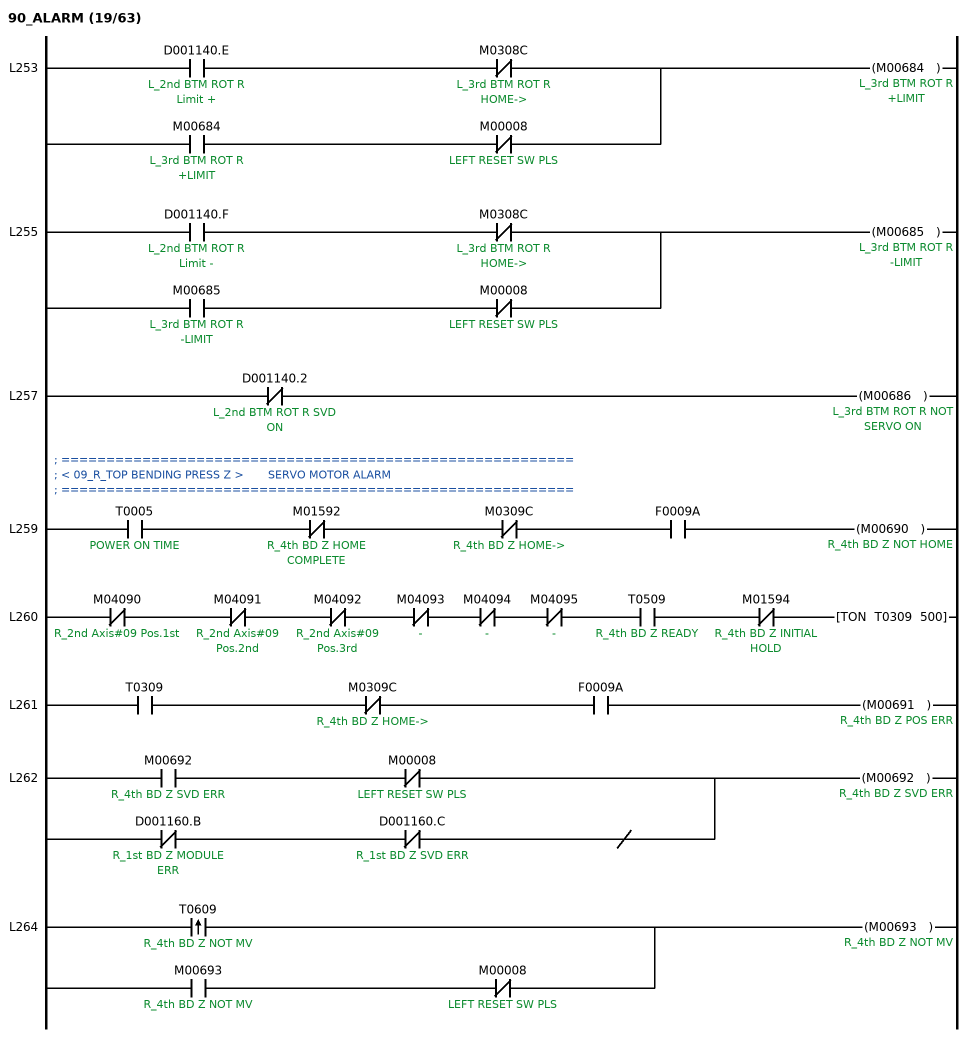
[picture p384: 90_ALARM rungs L253-L264]
; L253
LOAD      D001140.E	// L_2nd BTM ROT R Limit +
AND NOT   M0308C	// L_3rd BTM ROT R HOME->
LOAD      M00684	// L_3rd BTM ROT R +LIMIT
AND NOT   M00008	// LEFT RESET SW PLS
OR LOAD
OUT       M00684	// L_3rd BTM ROT R +LIMIT
; L255
LOAD      D001140.F	// L_2nd BTM ROT R Limit -
AND NOT   M0308C	// L_3rd BTM ROT R HOME->
LOAD      M00685	// L_3rd BTM ROT R -LIMIT
AND NOT   M00008	// LEFT RESET SW PLS
OR LOAD
OUT       M00685	// L_3rd BTM ROT R -LIMIT
; L257
LOAD NOT  D001140.2	// L_2nd BTM ROT R SVD ON
OUT       M00686	// L_3rd BTM ROT R NOT SERVO ON
// =========================================================
// 
//        < 09_R_TOP BENDING PRESS Z >       SERVO MOTOR ALARM
// 
// =========================================================
; L259
LOAD      T0005	// POWER ON TIME
AND NOT   M01592	// R_4th BD Z HOME COMPLETE
AND NOT   M0309C	// R_4th BD Z HOME->
AND       F0009A
OUT       M00690	// R_4th BD Z NOT HOME
; L260
LOAD NOT  M04090	// R_2nd Axis#09 Pos.1st
AND NOT   M04091	// R_2nd Axis#09 Pos.2nd
AND NOT   M04092	// R_2nd Axis#09 Pos.3rd
AND NOT   M04093	// -
AND NOT   M04094	// -
AND NOT   M04095	// -
AND       T0509	// R_4th BD Z READY
AND NOT   M01594	// R_4th BD Z INITIAL HOLD
TON       T0309 500
; L261
LOAD      T0309
AND NOT   M0309C	// R_4th BD Z HOME->
AND       F0009A
OUT       M00691	// R_4th BD Z POS ERR
; L262
LOAD      M00692	// R_4th BD Z SVD ERR
AND NOT   M00008	// LEFT RESET SW PLS
LOAD NOT  D001160.B	// R_1st BD Z MODULE ERR
AND NOT   D001160.C	// R_1st BD Z SVD ERR
NOT
OR LOAD
OUT       M00692	// R_4th BD Z SVD ERR
; L264
LOADP     T0609	// R_4th BD Z NOT MV
LOAD      M00693	// R_4th BD Z NOT MV
AND NOT   M00008	// LEFT RESET SW PLS
OR LOAD
OUT       M00693	// R_4th BD Z NOT MV

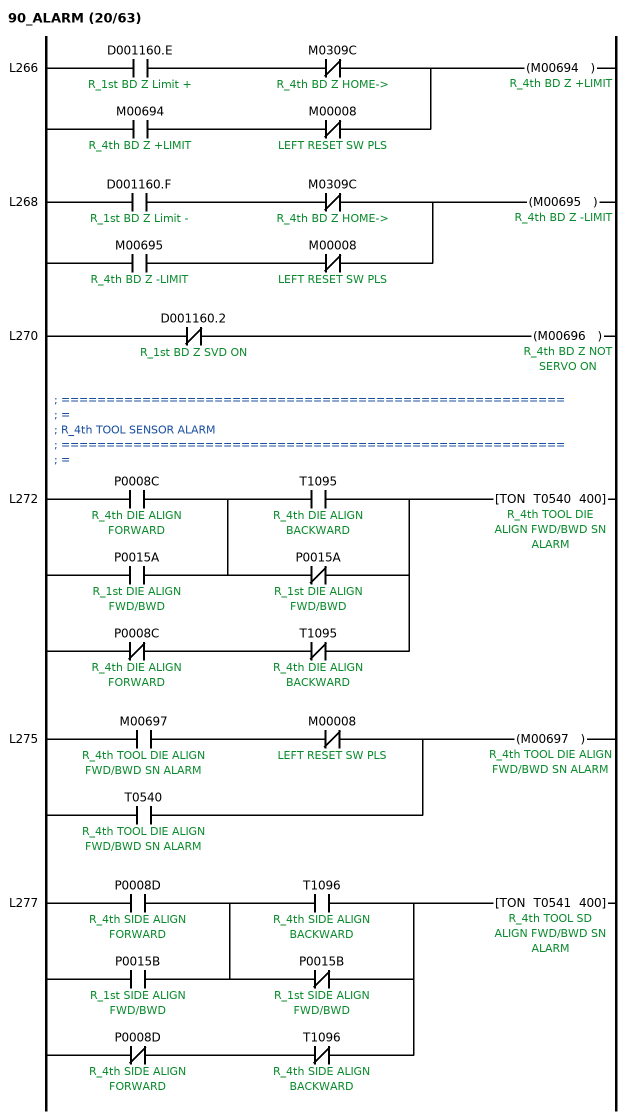
; L266
LOAD      D001160.E	// R_1st BD Z Limit +
AND NOT   M0309C	// R_4th BD Z HOME->
LOAD      M00694	// R_4th BD Z +LIMIT
AND NOT   M00008	// LEFT RESET SW PLS
OR LOAD
OUT       M00694	// R_4th BD Z +LIMIT
; L268
LOAD      D001160.F	// R_1st BD Z Limit -
AND NOT   M0309C	// R_4th BD Z HOME->
LOAD      M00695	// R_4th BD Z -LIMIT
AND NOT   M00008	// LEFT RESET SW PLS
OR LOAD
OUT       M00695	// R_4th BD Z -LIMIT
; L270
LOAD NOT  D001160.2	// R_1st BD Z SVD ON
OUT       M00696	// R_4th BD Z NOT SERVO ON
// =========================================================
// 
//        R_4th TOOL SENSOR ALARM
// 
// =========================================================
; L272
LOAD      P0008C	// R_4th DIE ALIGN FORWARD
OR        P0015A	// R_1st DIE ALIGN FWD/BWD
LOAD      T1095	// R_4th DIE ALIGN BACKWARD
OR NOT    P0015A	// R_1st DIE ALIGN FWD/BWD
AND LOAD
LOAD NOT  P0008C	// R_4th DIE ALIGN FORWARD
AND NOT   T1095	// R_4th DIE ALIGN BACKWARD
OR LOAD
TON       T0540 400	// R_4th TOOL DIE ALIGN FWD/BWD SN ALARM
; L275
LOAD      M00697	// R_4th TOOL DIE ALIGN FWD/BWD SN ALARM
AND NOT   M00008	// LEFT RESET SW PLS
OR        T0540	// R_4th TOOL DIE ALIGN FWD/BWD SN ALARM
OUT       M00697	// R_4th TOOL DIE ALIGN FWD/BWD SN ALARM
; L277
LOAD      P0008D	// R_4th SIDE ALIGN FORWARD
OR        P0015B	// R_1st SIDE ALIGN FWD/BWD
LOAD      T1096	// R_4th SIDE ALIGN BACKWARD
OR NOT    P0015B	// R_1st SIDE ALIGN FWD/BWD
AND LOAD
LOAD NOT  P0008D	// R_4th SIDE ALIGN FORWARD
AND NOT   T1096	// R_4th SIDE ALIGN BACKWARD
OR LOAD
TON       T0541 400	// R_4th TOOL SD ALIGN FWD/BWD SN ALARM

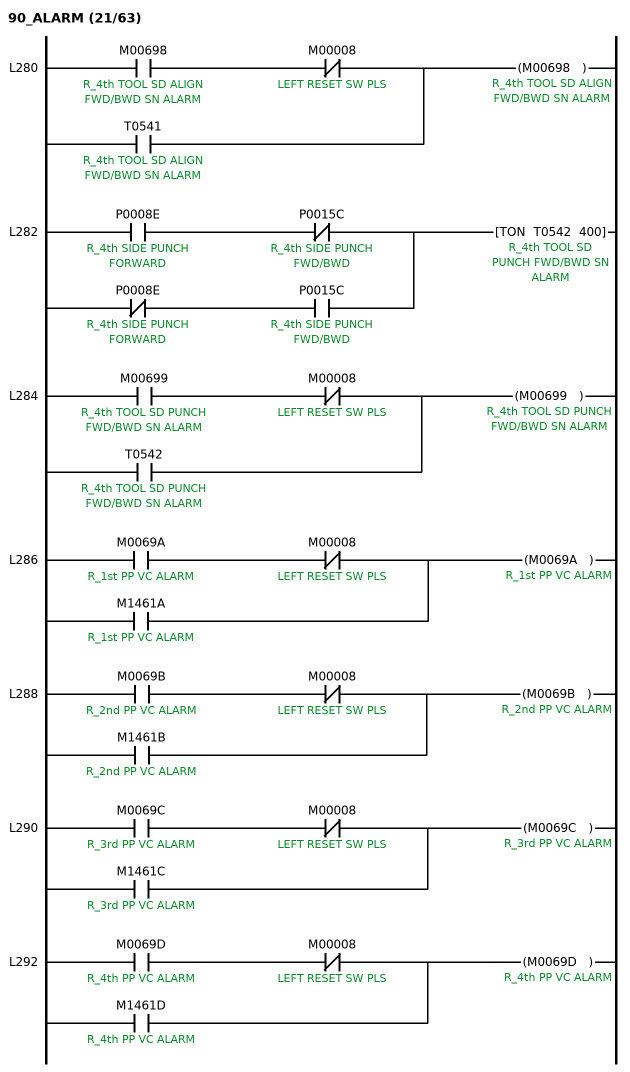
; L280
LOAD      M00698	// R_4th TOOL SD ALIGN FWD/BWD SN ALARM
AND NOT   M00008	// LEFT RESET SW PLS
OR        T0541	// R_4th TOOL SD ALIGN FWD/BWD SN ALARM
OUT       M00698	// R_4th TOOL SD ALIGN FWD/BWD SN ALARM
; L282
LOAD      P0008E	// R_4th SIDE PUNCH FORWARD
AND NOT   P0015C	// R_4th SIDE PUNCH FWD/BWD
LOAD NOT  P0008E	// R_4th SIDE PUNCH FORWARD
AND       P0015C	// R_4th SIDE PUNCH FWD/BWD
OR LOAD
TON       T0542 400	// R_4th TOOL SD PUNCH FWD/BWD SN ALARM
; L284
LOAD      M00699	// R_4th TOOL SD PUNCH FWD/BWD SN ALARM
AND NOT   M00008	// LEFT RESET SW PLS
OR        T0542	// R_4th TOOL SD PUNCH FWD/BWD SN ALARM
OUT       M00699	// R_4th TOOL SD PUNCH FWD/BWD SN ALARM
; L286
LOAD      M0069A	// R_1st PP VC ALARM
AND NOT   M00008	// LEFT RESET SW PLS
OR        M1461A	// R_1st PP VC ALARM
OUT       M0069A	// R_1st PP VC ALARM
; L288
LOAD      M0069B	// R_2nd PP VC ALARM
AND NOT   M00008	// LEFT RESET SW PLS
OR        M1461B	// R_2nd PP VC ALARM
OUT       M0069B	// R_2nd PP VC ALARM
; L290
LOAD      M0069C	// R_3rd PP VC ALARM
AND NOT   M00008	// LEFT RESET SW PLS
OR        M1461C	// R_3rd PP VC ALARM
OUT       M0069C	// R_3rd PP VC ALARM
; L292
LOAD      M0069D	// R_4th PP VC ALARM
AND NOT   M00008	// LEFT RESET SW PLS
OR        M1461D	// R_4th PP VC ALARM
OUT       M0069D	// R_4th PP VC ALARM

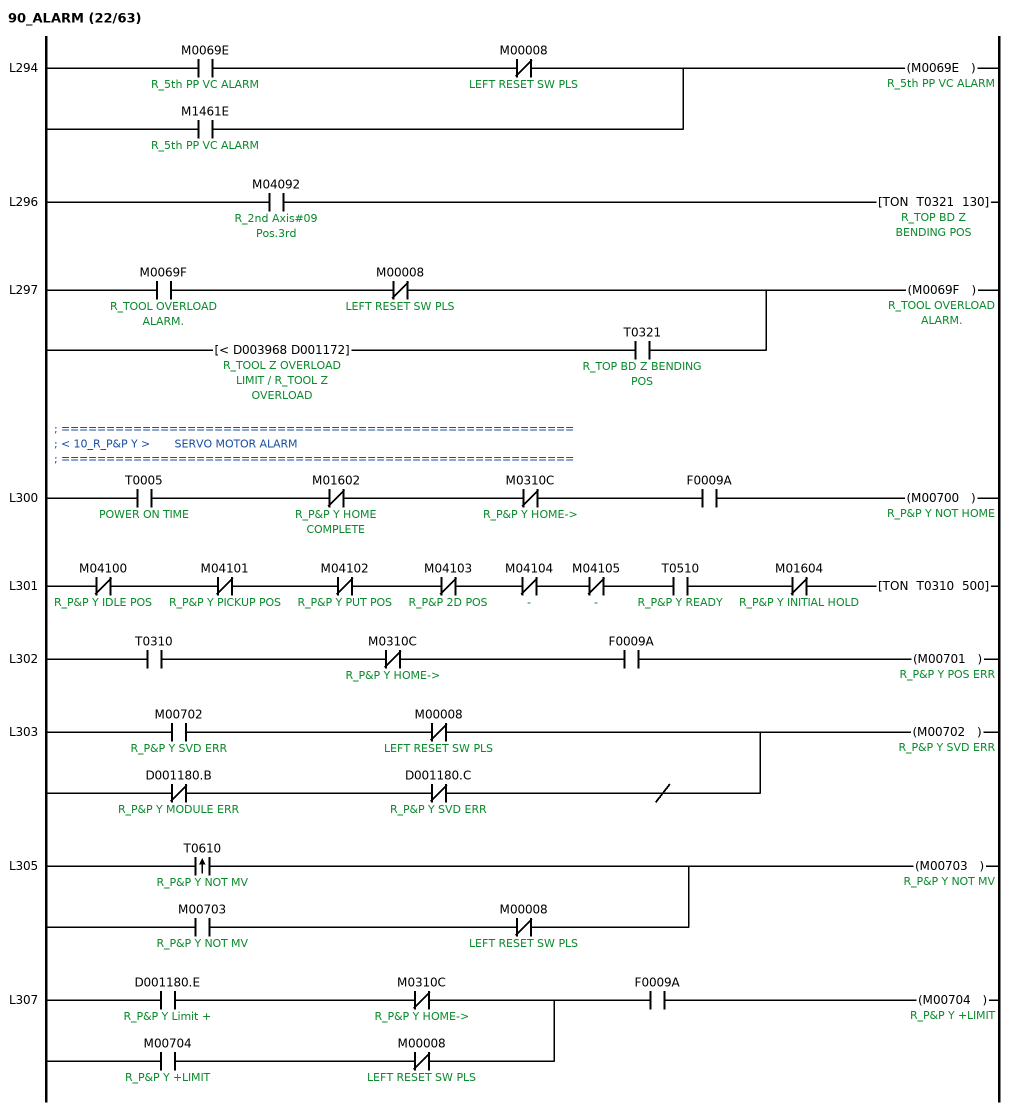
; L294
LOAD      M0069E	// R_5th PP VC ALARM
AND NOT   M00008	// LEFT RESET SW PLS
OR        M1461E	// R_5th PP VC ALARM
OUT       M0069E	// R_5th PP VC ALARM
; L296
LOAD      M04092	// R_2nd Axis#09 Pos.3rd
TON       T0321 130	// R_TOP BD Z BENDING POS
; L297
LOAD      M0069F	// R_TOOL OVERLOAD ALARM.
AND NOT   M00008	// LEFT RESET SW PLS
LOAD<     D003968 D001172	// R_TOOL Z OVERLOAD LIMIT / R_TOOL Z OVERLOAD
AND       T0321	// R_TOP BD Z BENDING POS
OR LOAD
OUT       M0069F	// R_TOOL OVERLOAD ALARM.
// =========================================================
// 
//        < 10_R_P&P Y >       SERVO MOTOR ALARM
// 
// =========================================================
; L300
LOAD      T0005	// POWER ON TIME
AND NOT   M01602	// R_P&P Y HOME COMPLETE
AND NOT   M0310C	// R_P&P Y HOME->
AND       F0009A
OUT       M00700	// R_P&P Y NOT HOME
; L301
LOAD NOT  M04100	// R_P&P Y IDLE POS
AND NOT   M04101	// R_P&P Y PICKUP POS
AND NOT   M04102	// R_P&P Y PUT POS
AND NOT   M04103	// R_P&P 2D POS
AND NOT   M04104	// -
AND NOT   M04105	// -
AND       T0510	// R_P&P Y READY
AND NOT   M01604	// R_P&P Y INITIAL HOLD
TON       T0310 500
; L302
LOAD      T0310
AND NOT   M0310C	// R_P&P Y HOME->
AND       F0009A
OUT       M00701	// R_P&P Y POS ERR
; L303
LOAD      M00702	// R_P&P Y SVD ERR
AND NOT   M00008	// LEFT RESET SW PLS
LOAD NOT  D001180.B	// R_P&P Y MODULE ERR
AND NOT   D001180.C	// R_P&P Y SVD ERR
NOT
OR LOAD
OUT       M00702	// R_P&P Y SVD ERR
; L305
LOADP     T0610	// R_P&P Y NOT MV
LOAD      M00703	// R_P&P Y NOT MV
AND NOT   M00008	// LEFT RESET SW PLS
OR LOAD
OUT       M00703	// R_P&P Y NOT MV
; L307
LOAD      D001180.E	// R_P&P Y Limit +
AND NOT   M0310C	// R_P&P Y HOME->
LOAD      M00704	// R_P&P Y +LIMIT
AND NOT   M00008	// LEFT RESET SW PLS
OR LOAD
AND       F0009A
OUT       M00704	// R_P&P Y +LIMIT

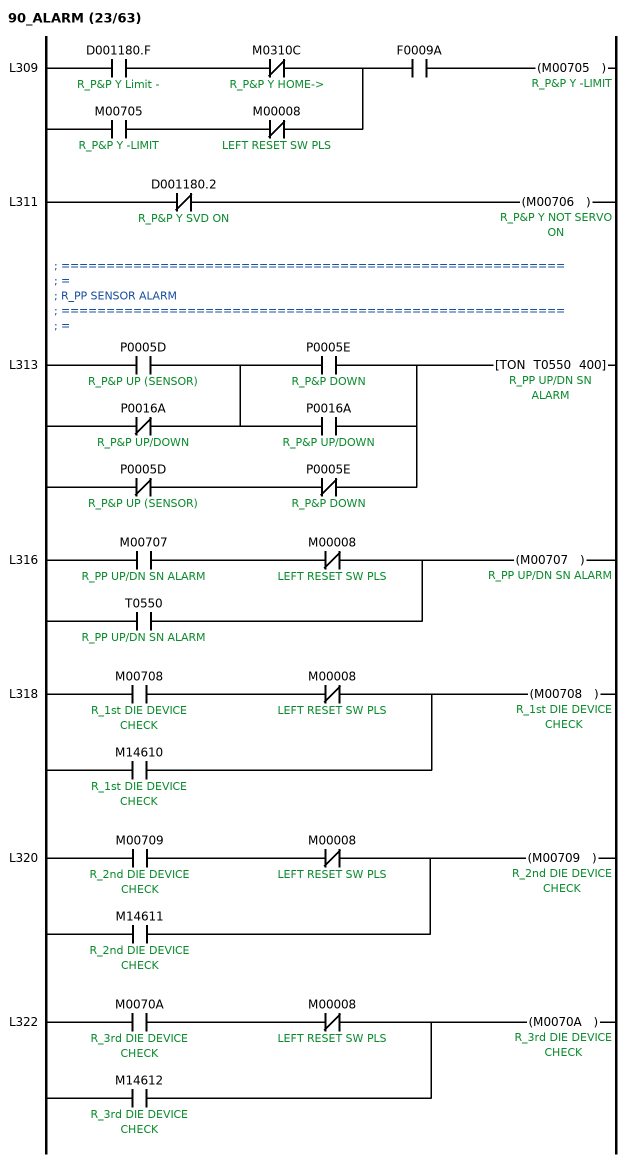
; L309
LOAD      D001180.F	// R_P&P Y Limit -
AND NOT   M0310C	// R_P&P Y HOME->
LOAD      M00705	// R_P&P Y -LIMIT
AND NOT   M00008	// LEFT RESET SW PLS
OR LOAD
AND       F0009A
OUT       M00705	// R_P&P Y -LIMIT
; L311
LOAD NOT  D001180.2	// R_P&P Y SVD ON
OUT       M00706	// R_P&P Y NOT SERVO ON
// =========================================================
// 
//       R_PP SENSOR ALARM
// 
// =========================================================
; L313
LOAD      P0005D	// R_P&P UP (SENSOR)
OR NOT    P0016A	// R_P&P UP/DOWN
LOAD      P0005E	// R_P&P DOWN
OR        P0016A	// R_P&P UP/DOWN
AND LOAD
LOAD NOT  P0005D	// R_P&P UP (SENSOR)
AND NOT   P0005E	// R_P&P DOWN
OR LOAD
TON       T0550 400	// R_PP UP/DN SN ALARM
; L316
LOAD      M00707	// R_PP UP/DN SN ALARM
AND NOT   M00008	// LEFT RESET SW PLS
OR        T0550	// R_PP UP/DN SN ALARM
OUT       M00707	// R_PP UP/DN SN ALARM
; L318
LOAD      M00708	// R_1st DIE DEVICE CHECK
AND NOT   M00008	// LEFT RESET SW PLS
OR        M14610	// R_1st DIE DEVICE CHECK
OUT       M00708	// R_1st DIE DEVICE CHECK
; L320
LOAD      M00709	// R_2nd DIE DEVICE CHECK
AND NOT   M00008	// LEFT RESET SW PLS
OR        M14611	// R_2nd DIE DEVICE CHECK
OUT       M00709	// R_2nd DIE DEVICE CHECK
; L322
LOAD      M0070A	// R_3rd DIE DEVICE CHECK
AND NOT   M00008	// LEFT RESET SW PLS
OR        M14612	// R_3rd DIE DEVICE CHECK
OUT       M0070A	// R_3rd DIE DEVICE CHECK

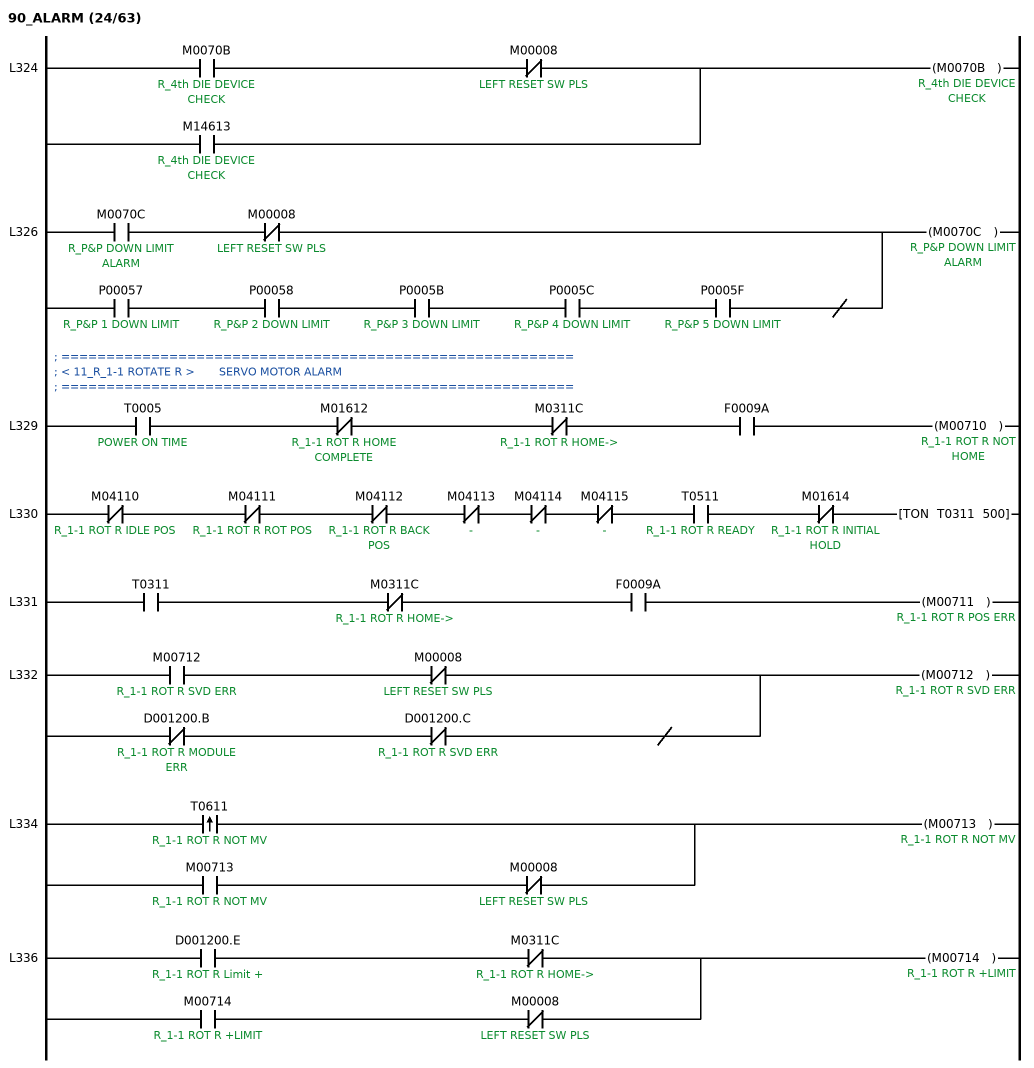
; L324
LOAD      M0070B	// R_4th DIE DEVICE CHECK
AND NOT   M00008	// LEFT RESET SW PLS
OR        M14613	// R_4th DIE DEVICE CHECK
OUT       M0070B	// R_4th DIE DEVICE CHECK
; L326
LOAD      M0070C	// R_P&P DOWN LIMIT ALARM
AND NOT   M00008	// LEFT RESET SW PLS
LOAD      P00057	// R_P&P 1 DOWN LIMIT
AND       P00058	// R_P&P 2 DOWN LIMIT
AND       P0005B	// R_P&P 3 DOWN LIMIT
AND       P0005C	// R_P&P 4 DOWN LIMIT
AND       P0005F	// R_P&P 5 DOWN LIMIT
NOT
OR LOAD
OUT       M0070C	// R_P&P DOWN LIMIT ALARM
// =========================================================
// 
//        < 11_R_1-1 ROTATE R >       SERVO MOTOR ALARM
// 
// =========================================================
; L329
LOAD      T0005	// POWER ON TIME
AND NOT   M01612	// R_1-1 ROT R HOME COMPLETE
AND NOT   M0311C	// R_1-1 ROT R HOME->
AND       F0009A
OUT       M00710	// R_1-1 ROT R NOT HOME
; L330
LOAD NOT  M04110	// R_1-1 ROT R IDLE POS
AND NOT   M04111	// R_1-1 ROT R ROT POS
AND NOT   M04112	// R_1-1 ROT R BACK POS
AND NOT   M04113	// -
AND NOT   M04114	// -
AND NOT   M04115	// -
AND       T0511	// R_1-1 ROT R READY
AND NOT   M01614	// R_1-1 ROT R INITIAL HOLD
TON       T0311 500
; L331
LOAD      T0311
AND NOT   M0311C	// R_1-1 ROT R HOME->
AND       F0009A
OUT       M00711	// R_1-1 ROT R POS ERR
; L332
LOAD      M00712	// R_1-1 ROT R SVD ERR
AND NOT   M00008	// LEFT RESET SW PLS
LOAD NOT  D001200.B	// R_1-1 ROT R MODULE ERR
AND NOT   D001200.C	// R_1-1 ROT R SVD ERR
NOT
OR LOAD
OUT       M00712	// R_1-1 ROT R SVD ERR
; L334
LOADP     T0611	// R_1-1 ROT R NOT MV
LOAD      M00713	// R_1-1 ROT R NOT MV
AND NOT   M00008	// LEFT RESET SW PLS
OR LOAD
OUT       M00713	// R_1-1 ROT R NOT MV
; L336
LOAD      D001200.E	// R_1-1 ROT R Limit +
AND NOT   M0311C	// R_1-1 ROT R HOME->
LOAD      M00714	// R_1-1 ROT R +LIMIT
AND NOT   M00008	// LEFT RESET SW PLS
OR LOAD
OUT       M00714	// R_1-1 ROT R +LIMIT

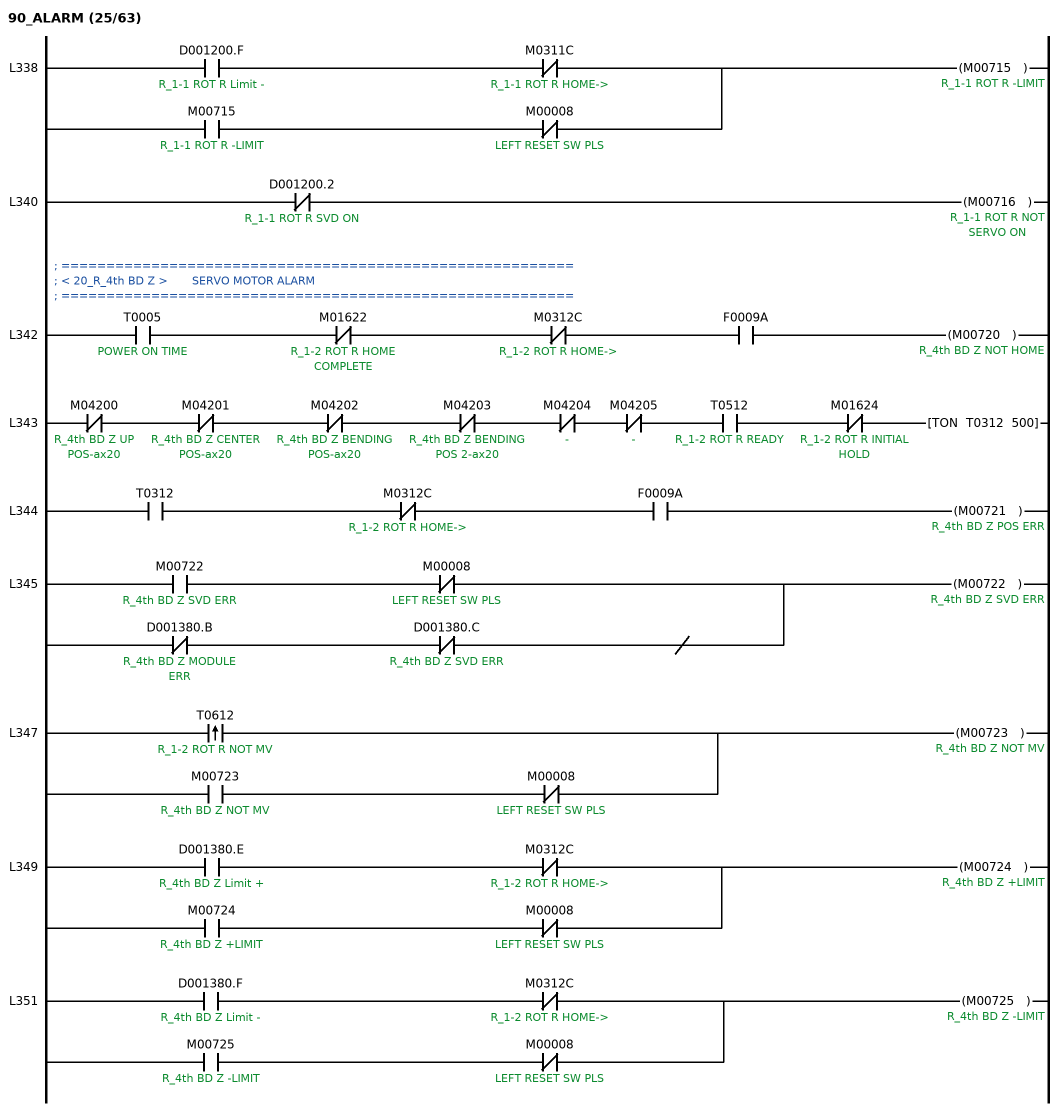
; L338
LOAD      D001200.F	// R_1-1 ROT R Limit -
AND NOT   M0311C	// R_1-1 ROT R HOME->
LOAD      M00715	// R_1-1 ROT R -LIMIT
AND NOT   M00008	// LEFT RESET SW PLS
OR LOAD
OUT       M00715	// R_1-1 ROT R -LIMIT
; L340
LOAD NOT  D001200.2	// R_1-1 ROT R SVD ON
OUT       M00716	// R_1-1 ROT R NOT SERVO ON
// =========================================================
// 
//        < 20_R_4th BD Z >       SERVO MOTOR ALARM
// 
// =========================================================
; L342
LOAD      T0005	// POWER ON TIME
AND NOT   M01622	// R_1-2 ROT R HOME COMPLETE
AND NOT   M0312C	// R_1-2 ROT R HOME->
AND       F0009A
OUT       M00720	// R_4th BD Z NOT HOME
; L343
LOAD NOT  M04200	// R_4th BD Z UP POS-ax20
AND NOT   M04201	// R_4th BD Z CENTER POS-ax20
AND NOT   M04202	// R_4th BD Z BENDING POS-ax20
AND NOT   M04203	// R_4th BD Z BENDING POS 2-ax20
AND NOT   M04204	// -
AND NOT   M04205	// -
AND       T0512	// R_1-2 ROT R READY
AND NOT   M01624	// R_1-2 ROT R INITIAL HOLD
TON       T0312 500
; L344
LOAD      T0312
AND NOT   M0312C	// R_1-2 ROT R HOME->
AND       F0009A
OUT       M00721	// R_4th BD Z POS ERR
; L345
LOAD      M00722	// R_4th BD Z SVD ERR
AND NOT   M00008	// LEFT RESET SW PLS
LOAD NOT  D001380.B	// R_4th BD Z MODULE ERR
AND NOT   D001380.C	// R_4th BD Z SVD ERR
NOT
OR LOAD
OUT       M00722	// R_4th BD Z SVD ERR
; L347
LOADP     T0612	// R_1-2 ROT R NOT MV
LOAD      M00723	// R_4th BD Z NOT MV
AND NOT   M00008	// LEFT RESET SW PLS
OR LOAD
OUT       M00723	// R_4th BD Z NOT MV
; L349
LOAD      D001380.E	// R_4th BD Z Limit +
AND NOT   M0312C	// R_1-2 ROT R HOME->
LOAD      M00724	// R_4th BD Z +LIMIT
AND NOT   M00008	// LEFT RESET SW PLS
OR LOAD
OUT       M00724	// R_4th BD Z +LIMIT
; L351
LOAD      D001380.F	// R_4th BD Z Limit -
AND NOT   M0312C	// R_1-2 ROT R HOME->
LOAD      M00725	// R_4th BD Z -LIMIT
AND NOT   M00008	// LEFT RESET SW PLS
OR LOAD
OUT       M00725	// R_4th BD Z -LIMIT

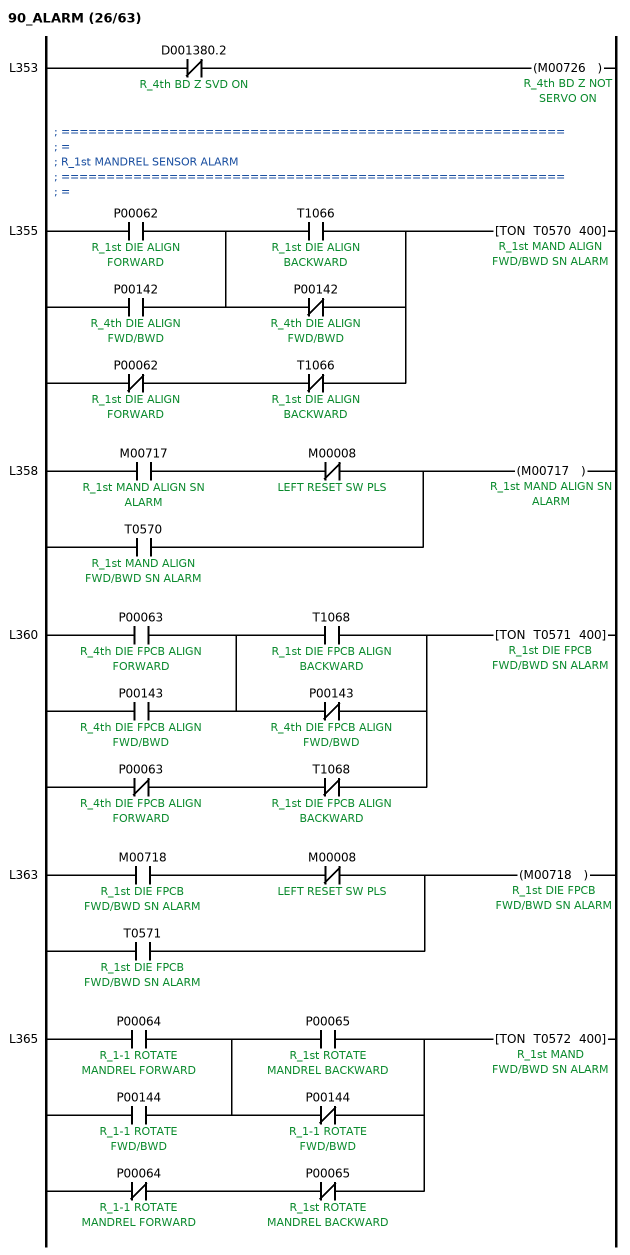
; L353
LOAD NOT  D001380.2	// R_4th BD Z SVD ON
OUT       M00726	// R_4th BD Z NOT SERVO ON
// =========================================================
// 
//        R_1st MANDREL SENSOR ALARM
// 
// =========================================================
; L355
LOAD      P00062	// R_1st DIE ALIGN FORWARD
OR        P00142	// R_4th DIE ALIGN FWD/BWD
LOAD      T1066	// R_1st DIE ALIGN BACKWARD
OR NOT    P00142	// R_4th DIE ALIGN FWD/BWD
AND LOAD
LOAD NOT  P00062	// R_1st DIE ALIGN FORWARD
AND NOT   T1066	// R_1st DIE ALIGN BACKWARD
OR LOAD
TON       T0570 400	// R_1st MAND ALIGN FWD/BWD SN ALARM
; L358
LOAD      M00717	// R_1st MAND ALIGN SN ALARM
AND NOT   M00008	// LEFT RESET SW PLS
OR        T0570	// R_1st MAND ALIGN FWD/BWD SN ALARM
OUT       M00717	// R_1st MAND ALIGN SN ALARM
; L360
LOAD      P00063	// R_4th DIE FPCB ALIGN FORWARD
OR        P00143	// R_4th DIE FPCB ALIGN FWD/BWD
LOAD      T1068	// R_1st DIE FPCB ALIGN BACKWARD
OR NOT    P00143	// R_4th DIE FPCB ALIGN FWD/BWD
AND LOAD
LOAD NOT  P00063	// R_4th DIE FPCB ALIGN FORWARD
AND NOT   T1068	// R_1st DIE FPCB ALIGN BACKWARD
OR LOAD
TON       T0571 400	// R_1st DIE FPCB FWD/BWD SN ALARM
; L363
LOAD      M00718	// R_1st DIE FPCB FWD/BWD SN ALARM
AND NOT   M00008	// LEFT RESET SW PLS
OR        T0571	// R_1st DIE FPCB FWD/BWD SN ALARM
OUT       M00718	// R_1st DIE FPCB FWD/BWD SN ALARM
; L365
LOAD      P00064	// R_1-1 ROTATE MANDREL FORWARD
OR        P00144	// R_1-1 ROTATE FWD/BWD
LOAD      P00065	// R_1st ROTATE MANDREL BACKWARD
OR NOT    P00144	// R_1-1 ROTATE FWD/BWD
AND LOAD
LOAD NOT  P00064	// R_1-1 ROTATE MANDREL FORWARD
AND NOT   P00065	// R_1st ROTATE MANDREL BACKWARD
OR LOAD
TON       T0572 400	// R_1st MAND FWD/BWD SN ALARM

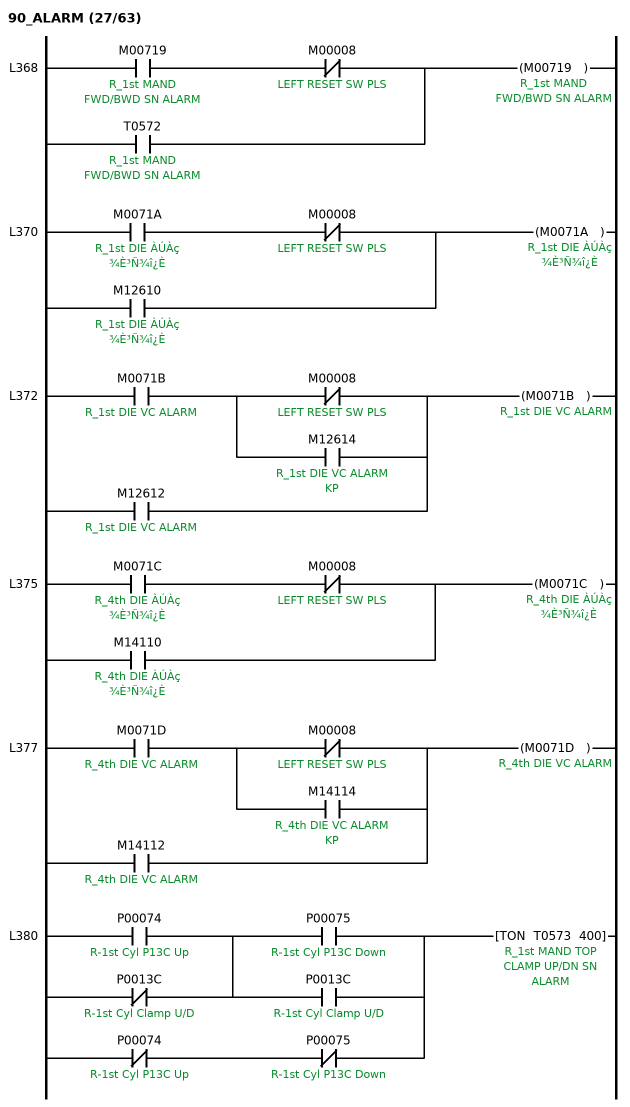
; L368
LOAD      M00719	// R_1st MAND FWD/BWD SN ALARM
AND NOT   M00008	// LEFT RESET SW PLS
OR        T0572	// R_1st MAND FWD/BWD SN ALARM
OUT       M00719	// R_1st MAND FWD/BWD SN ALARM
; L370
LOAD      M0071A	// R_1st DIE ÀÚÀç ¾È³Ñ¾î¿È
AND NOT   M00008	// LEFT RESET SW PLS
OR        M12610	// R_1st DIE ÀÚÀç ¾È³Ñ¾î¿È
OUT       M0071A	// R_1st DIE ÀÚÀç ¾È³Ñ¾î¿È
; L372
LOAD      M0071B	// R_1st DIE VC ALARM
LOAD NOT  M00008	// LEFT RESET SW PLS
OR        M12614	// R_1st DIE VC ALARM KP
AND LOAD
OR        M12612	// R_1st DIE VC ALARM
OUT       M0071B	// R_1st DIE VC ALARM
; L375
LOAD      M0071C	// R_4th DIE ÀÚÀç ¾È³Ñ¾î¿È
AND NOT   M00008	// LEFT RESET SW PLS
OR        M14110	// R_4th DIE ÀÚÀç ¾È³Ñ¾î¿È
OUT       M0071C	// R_4th DIE ÀÚÀç ¾È³Ñ¾î¿È
; L377
LOAD      M0071D	// R_4th DIE VC ALARM
LOAD NOT  M00008	// LEFT RESET SW PLS
OR        M14114	// R_4th DIE VC ALARM KP
AND LOAD
OR        M14112	// R_4th DIE VC ALARM
OUT       M0071D	// R_4th DIE VC ALARM
; L380
LOAD      P00074	// R-1st Cyl P13C Up
OR NOT    P0013C	// R-1st Cyl Clamp U/D
LOAD      P00075	// R-1st Cyl P13C Down
OR        P0013C	// R-1st Cyl Clamp U/D
AND LOAD
LOAD NOT  P00074	// R-1st Cyl P13C Up
AND NOT   P00075	// R-1st Cyl P13C Down
OR LOAD
TON       T0573 400	// R_1st MAND TOP CLAMP UP/DN SN ALARM

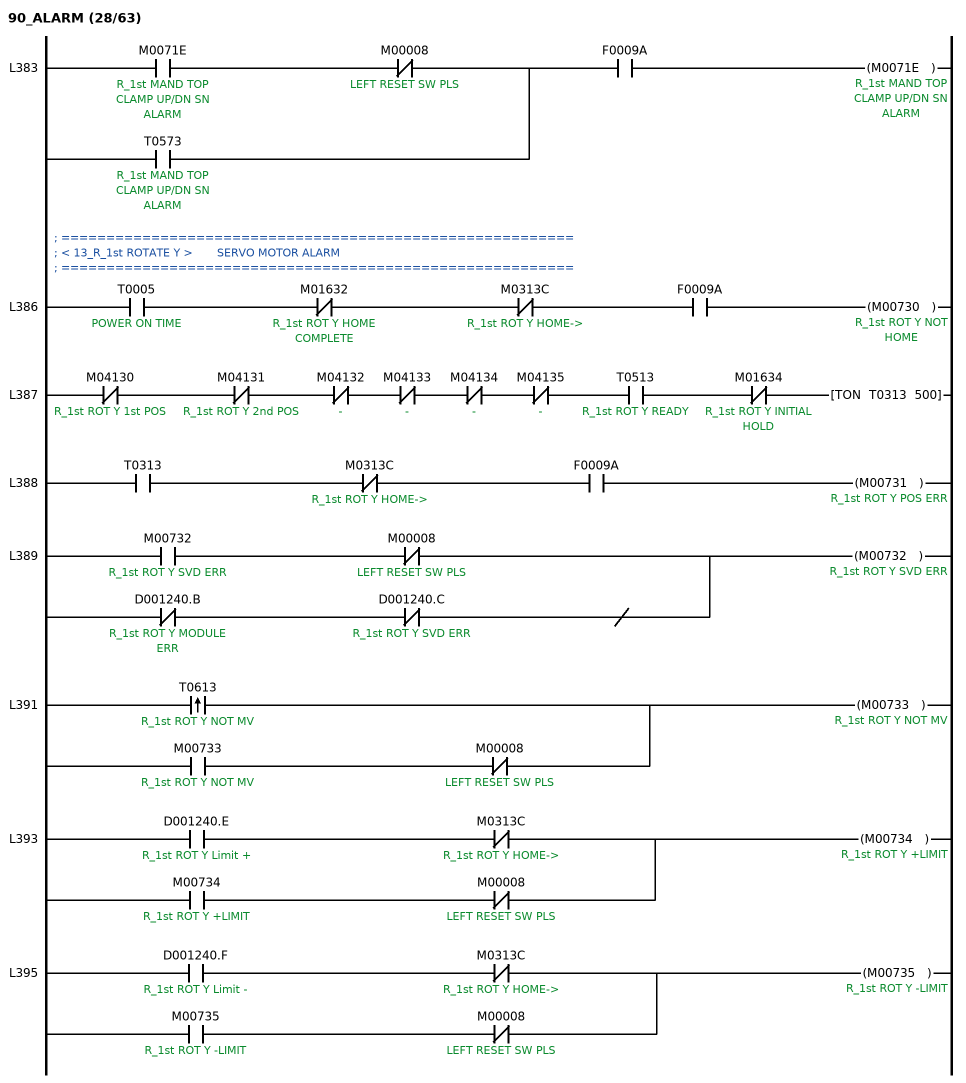
; L383
LOAD      M0071E	// R_1st MAND TOP CLAMP UP/DN SN ALARM
AND NOT   M00008	// LEFT RESET SW PLS
OR        T0573	// R_1st MAND TOP CLAMP UP/DN SN ALARM
AND       F0009A
OUT       M0071E	// R_1st MAND TOP CLAMP UP/DN SN ALARM
// =========================================================
// 
//        < 13_R_1st ROTATE Y >       SERVO MOTOR ALARM
// 
// =========================================================
; L386
LOAD      T0005	// POWER ON TIME
AND NOT   M01632	// R_1st ROT Y HOME COMPLETE
AND NOT   M0313C	// R_1st ROT Y HOME->
AND       F0009A
OUT       M00730	// R_1st ROT Y NOT HOME
; L387
LOAD NOT  M04130	// R_1st ROT Y 1st POS
AND NOT   M04131	// R_1st ROT Y 2nd POS
AND NOT   M04132	// -
AND NOT   M04133	// -
AND NOT   M04134	// -
AND NOT   M04135	// -
AND       T0513	// R_1st ROT Y READY
AND NOT   M01634	// R_1st ROT Y INITIAL HOLD
TON       T0313 500
; L388
LOAD      T0313
AND NOT   M0313C	// R_1st ROT Y HOME->
AND       F0009A
OUT       M00731	// R_1st ROT Y POS ERR
; L389
LOAD      M00732	// R_1st ROT Y SVD ERR
AND NOT   M00008	// LEFT RESET SW PLS
LOAD NOT  D001240.B	// R_1st ROT Y MODULE ERR
AND NOT   D001240.C	// R_1st ROT Y SVD ERR
NOT
OR LOAD
OUT       M00732	// R_1st ROT Y SVD ERR
; L391
LOADP     T0613	// R_1st ROT Y NOT MV
LOAD      M00733	// R_1st ROT Y NOT MV
AND NOT   M00008	// LEFT RESET SW PLS
OR LOAD
OUT       M00733	// R_1st ROT Y NOT MV
; L393
LOAD      D001240.E	// R_1st ROT Y Limit +
AND NOT   M0313C	// R_1st ROT Y HOME->
LOAD      M00734	// R_1st ROT Y +LIMIT
AND NOT   M00008	// LEFT RESET SW PLS
OR LOAD
OUT       M00734	// R_1st ROT Y +LIMIT
; L395
LOAD      D001240.F	// R_1st ROT Y Limit -
AND NOT   M0313C	// R_1st ROT Y HOME->
LOAD      M00735	// R_1st ROT Y -LIMIT
AND NOT   M00008	// LEFT RESET SW PLS
OR LOAD
OUT       M00735	// R_1st ROT Y -LIMIT

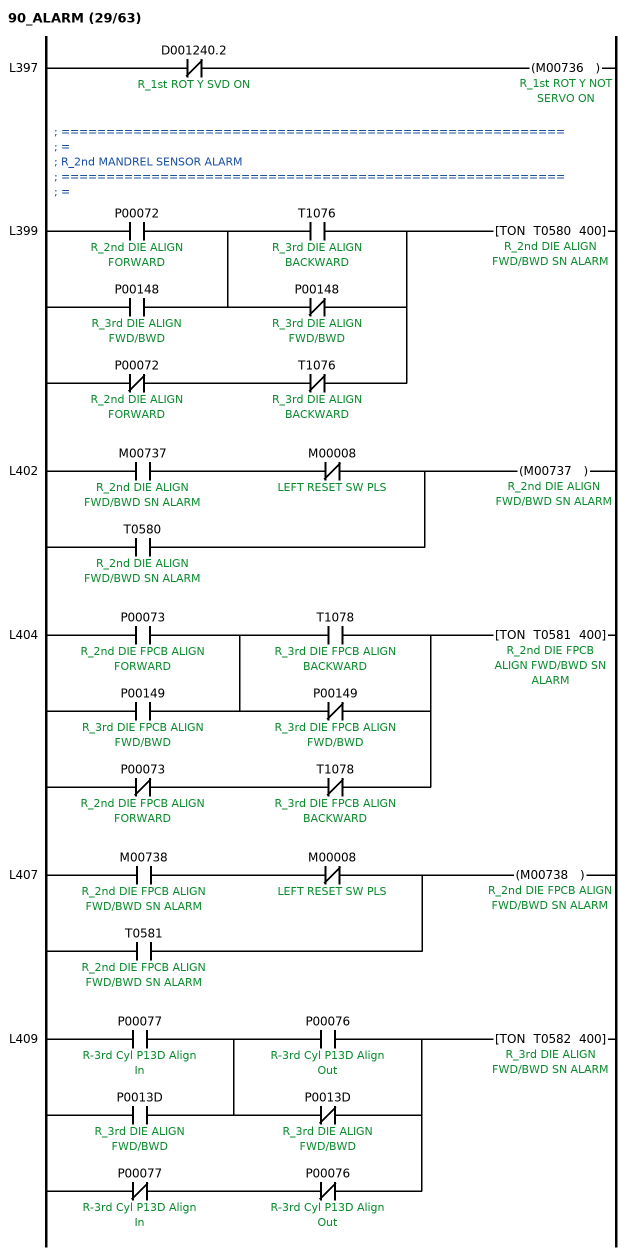
; L397
LOAD NOT  D001240.2	// R_1st ROT Y SVD ON
OUT       M00736	// R_1st ROT Y NOT SERVO ON
// =========================================================
// 
//        R_2nd MANDREL SENSOR ALARM
// 
// =========================================================
; L399
LOAD      P00072	// R_2nd DIE ALIGN FORWARD
OR        P00148	// R_3rd DIE ALIGN FWD/BWD
LOAD      T1076	// R_3rd DIE ALIGN BACKWARD
OR NOT    P00148	// R_3rd DIE ALIGN FWD/BWD
AND LOAD
LOAD NOT  P00072	// R_2nd DIE ALIGN FORWARD
AND NOT   T1076	// R_3rd DIE ALIGN BACKWARD
OR LOAD
TON       T0580 400	// R_2nd DIE ALIGN FWD/BWD SN ALARM
; L402
LOAD      M00737	// R_2nd DIE ALIGN FWD/BWD SN ALARM
AND NOT   M00008	// LEFT RESET SW PLS
OR        T0580	// R_2nd DIE ALIGN FWD/BWD SN ALARM
OUT       M00737	// R_2nd DIE ALIGN FWD/BWD SN ALARM
; L404
LOAD      P00073	// R_2nd DIE FPCB ALIGN FORWARD
OR        P00149	// R_3rd DIE FPCB ALIGN FWD/BWD
LOAD      T1078	// R_3rd DIE FPCB ALIGN BACKWARD
OR NOT    P00149	// R_3rd DIE FPCB ALIGN FWD/BWD
AND LOAD
LOAD NOT  P00073	// R_2nd DIE FPCB ALIGN FORWARD
AND NOT   T1078	// R_3rd DIE FPCB ALIGN BACKWARD
OR LOAD
TON       T0581 400	// R_2nd DIE FPCB ALIGN FWD/BWD SN ALARM
; L407
LOAD      M00738	// R_2nd DIE FPCB ALIGN FWD/BWD SN ALARM
AND NOT   M00008	// LEFT RESET SW PLS
OR        T0581	// R_2nd DIE FPCB ALIGN FWD/BWD SN ALARM
OUT       M00738	// R_2nd DIE FPCB ALIGN FWD/BWD SN ALARM
; L409
LOAD      P00077	// R-3rd Cyl P13D Align In
OR        P0013D	// R_3rd DIE ALIGN FWD/BWD
LOAD      P00076	// R-3rd Cyl P13D Align Out
OR NOT    P0013D	// R_3rd DIE ALIGN FWD/BWD
AND LOAD
LOAD NOT  P00077	// R-3rd Cyl P13D Align In
AND NOT   P00076	// R-3rd Cyl P13D Align Out
OR LOAD
TON       T0582 400	// R_3rd DIE ALIGN FWD/BWD SN ALARM

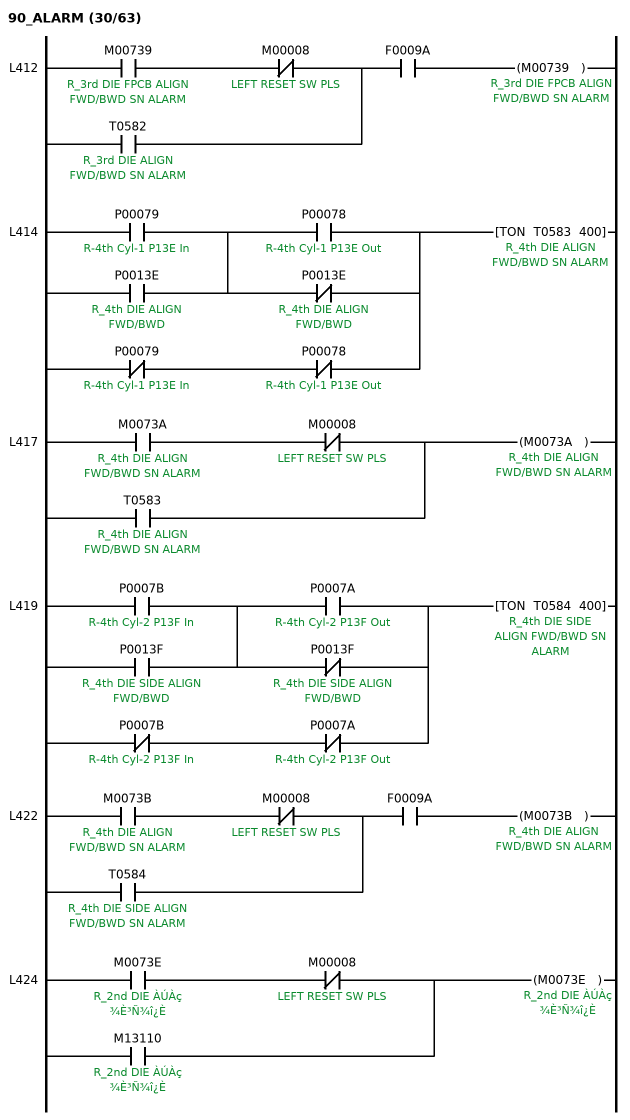
; L412
LOAD      M00739	// R_3rd DIE FPCB ALIGN FWD/BWD SN ALARM
AND NOT   M00008	// LEFT RESET SW PLS
OR        T0582	// R_3rd DIE ALIGN FWD/BWD SN ALARM
AND       F0009A
OUT       M00739	// R_3rd DIE FPCB ALIGN FWD/BWD SN ALARM
; L414
LOAD      P00079	// R-4th Cyl-1 P13E In
OR        P0013E	// R_4th DIE ALIGN FWD/BWD
LOAD      P00078	// R-4th Cyl-1 P13E Out
OR NOT    P0013E	// R_4th DIE ALIGN FWD/BWD
AND LOAD
LOAD NOT  P00079	// R-4th Cyl-1 P13E In
AND NOT   P00078	// R-4th Cyl-1 P13E Out
OR LOAD
TON       T0583 400	// R_4th DIE ALIGN FWD/BWD SN ALARM
; L417
LOAD      M0073A	// R_4th DIE ALIGN FWD/BWD SN ALARM
AND NOT   M00008	// LEFT RESET SW PLS
OR        T0583	// R_4th DIE ALIGN FWD/BWD SN ALARM
OUT       M0073A	// R_4th DIE ALIGN FWD/BWD SN ALARM
; L419
LOAD      P0007B	// R-4th Cyl-2 P13F In
OR        P0013F	// R_4th DIE SIDE ALIGN FWD/BWD
LOAD      P0007A	// R-4th Cyl-2 P13F Out
OR NOT    P0013F	// R_4th DIE SIDE ALIGN FWD/BWD
AND LOAD
LOAD NOT  P0007B	// R-4th Cyl-2 P13F In
AND NOT   P0007A	// R-4th Cyl-2 P13F Out
OR LOAD
TON       T0584 400	// R_4th DIE SIDE ALIGN FWD/BWD SN ALARM
; L422
LOAD      M0073B	// R_4th DIE ALIGN FWD/BWD SN ALARM
AND NOT   M00008	// LEFT RESET SW PLS
OR        T0584	// R_4th DIE SIDE ALIGN FWD/BWD SN ALARM
AND       F0009A
OUT       M0073B	// R_4th DIE ALIGN FWD/BWD SN ALARM
; L424
LOAD      M0073E	// R_2nd DIE ÀÚÀç ¾È³Ñ¾î¿È
AND NOT   M00008	// LEFT RESET SW PLS
OR        M13110	// R_2nd DIE ÀÚÀç ¾È³Ñ¾î¿È
OUT       M0073E	// R_2nd DIE ÀÚÀç ¾È³Ñ¾î¿È

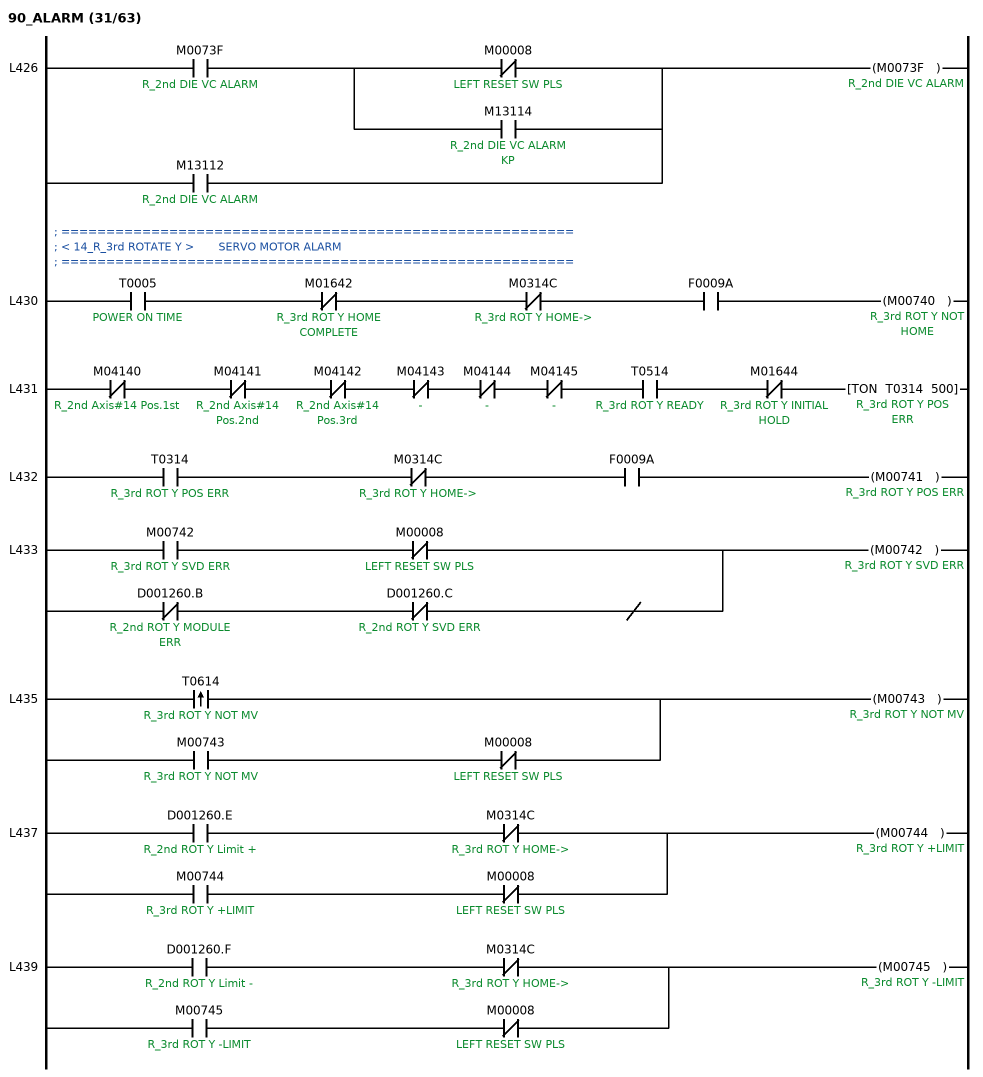
; L426
LOAD      M0073F	// R_2nd DIE VC ALARM
LOAD NOT  M00008	// LEFT RESET SW PLS
OR        M13114	// R_2nd DIE VC ALARM KP
AND LOAD
OR        M13112	// R_2nd DIE VC ALARM
OUT       M0073F	// R_2nd DIE VC ALARM
// =========================================================
// 
//        < 14_R_3rd ROTATE Y >       SERVO MOTOR ALARM
// 
// =========================================================
; L430
LOAD      T0005	// POWER ON TIME
AND NOT   M01642	// R_3rd ROT Y HOME COMPLETE
AND NOT   M0314C	// R_3rd ROT Y HOME->
AND       F0009A
OUT       M00740	// R_3rd ROT Y NOT HOME
; L431
LOAD NOT  M04140	// R_2nd Axis#14 Pos.1st
AND NOT   M04141	// R_2nd Axis#14 Pos.2nd
AND NOT   M04142	// R_2nd Axis#14 Pos.3rd
AND NOT   M04143	// -
AND NOT   M04144	// -
AND NOT   M04145	// -
AND       T0514	// R_3rd ROT Y READY
AND NOT   M01644	// R_3rd ROT Y INITIAL HOLD
TON       T0314 500	// R_3rd ROT Y POS ERR
; L432
LOAD      T0314	// R_3rd ROT Y POS ERR
AND NOT   M0314C	// R_3rd ROT Y HOME->
AND       F0009A
OUT       M00741	// R_3rd ROT Y POS ERR
; L433
LOAD      M00742	// R_3rd ROT Y SVD ERR
AND NOT   M00008	// LEFT RESET SW PLS
LOAD NOT  D001260.B	// R_2nd ROT Y MODULE ERR
AND NOT   D001260.C	// R_2nd ROT Y SVD ERR
NOT
OR LOAD
OUT       M00742	// R_3rd ROT Y SVD ERR
; L435
LOADP     T0614	// R_3rd ROT Y NOT MV
LOAD      M00743	// R_3rd ROT Y NOT MV
AND NOT   M00008	// LEFT RESET SW PLS
OR LOAD
OUT       M00743	// R_3rd ROT Y NOT MV
; L437
LOAD      D001260.E	// R_2nd ROT Y Limit +
AND NOT   M0314C	// R_3rd ROT Y HOME->
LOAD      M00744	// R_3rd ROT Y +LIMIT
AND NOT   M00008	// LEFT RESET SW PLS
OR LOAD
OUT       M00744	// R_3rd ROT Y +LIMIT
; L439
LOAD      D001260.F	// R_2nd ROT Y Limit -
AND NOT   M0314C	// R_3rd ROT Y HOME->
LOAD      M00745	// R_3rd ROT Y -LIMIT
AND NOT   M00008	// LEFT RESET SW PLS
OR LOAD
OUT       M00745	// R_3rd ROT Y -LIMIT

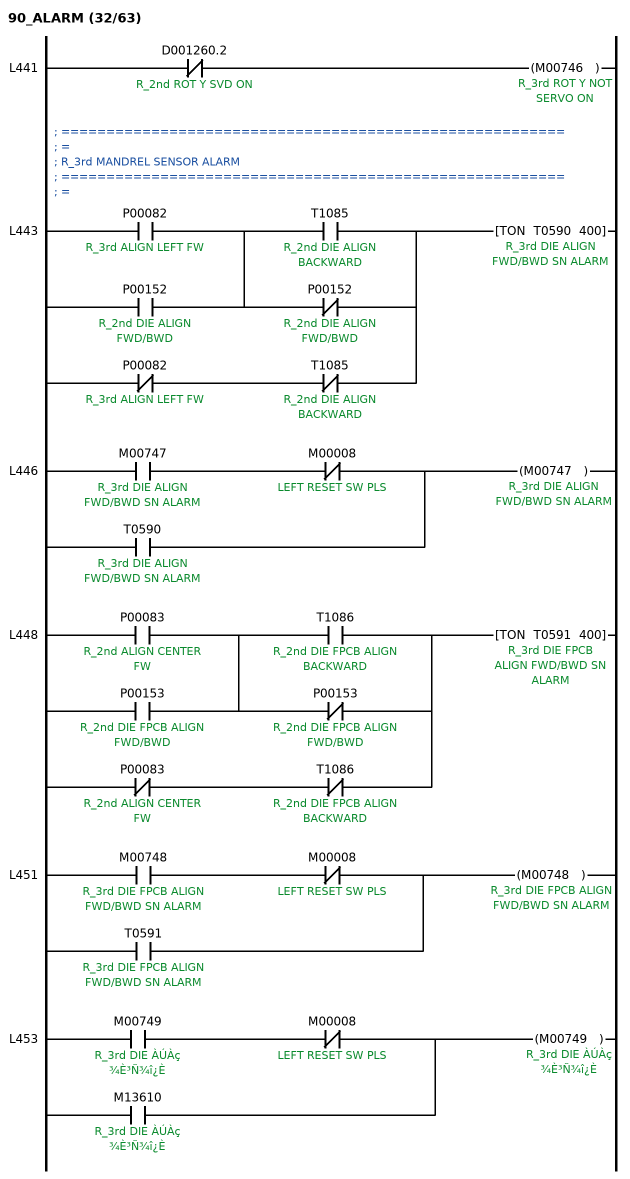
; L441
LOAD NOT  D001260.2	// R_2nd ROT Y SVD ON
OUT       M00746	// R_3rd ROT Y NOT SERVO ON
// =========================================================
// 
//        R_3rd MANDREL SENSOR ALARM
// 
// =========================================================
; L443
LOAD      P00082	// R_3rd ALIGN LEFT FW
OR        P00152	// R_2nd DIE ALIGN FWD/BWD
LOAD      T1085	// R_2nd DIE ALIGN BACKWARD
OR NOT    P00152	// R_2nd DIE ALIGN FWD/BWD
AND LOAD
LOAD NOT  P00082	// R_3rd ALIGN LEFT FW
AND NOT   T1085	// R_2nd DIE ALIGN BACKWARD
OR LOAD
TON       T0590 400	// R_3rd DIE ALIGN FWD/BWD SN ALARM
; L446
LOAD      M00747	// R_3rd DIE ALIGN FWD/BWD SN ALARM
AND NOT   M00008	// LEFT RESET SW PLS
OR        T0590	// R_3rd DIE ALIGN FWD/BWD SN ALARM
OUT       M00747	// R_3rd DIE ALIGN FWD/BWD SN ALARM
; L448
LOAD      P00083	// R_2nd ALIGN CENTER FW
OR        P00153	// R_2nd DIE FPCB ALIGN FWD/BWD
LOAD      T1086	// R_2nd DIE FPCB ALIGN BACKWARD
OR NOT    P00153	// R_2nd DIE FPCB ALIGN FWD/BWD
AND LOAD
LOAD NOT  P00083	// R_2nd ALIGN CENTER FW
AND NOT   T1086	// R_2nd DIE FPCB ALIGN BACKWARD
OR LOAD
TON       T0591 400	// R_3rd DIE FPCB ALIGN FWD/BWD SN ALARM
; L451
LOAD      M00748	// R_3rd DIE FPCB ALIGN FWD/BWD SN ALARM
AND NOT   M00008	// LEFT RESET SW PLS
OR        T0591	// R_3rd DIE FPCB ALIGN FWD/BWD SN ALARM
OUT       M00748	// R_3rd DIE FPCB ALIGN FWD/BWD SN ALARM
; L453
LOAD      M00749	// R_3rd DIE ÀÚÀç ¾È³Ñ¾î¿È
AND NOT   M00008	// LEFT RESET SW PLS
OR        M13610	// R_3rd DIE ÀÚÀç ¾È³Ñ¾î¿È
OUT       M00749	// R_3rd DIE ÀÚÀç ¾È³Ñ¾î¿È

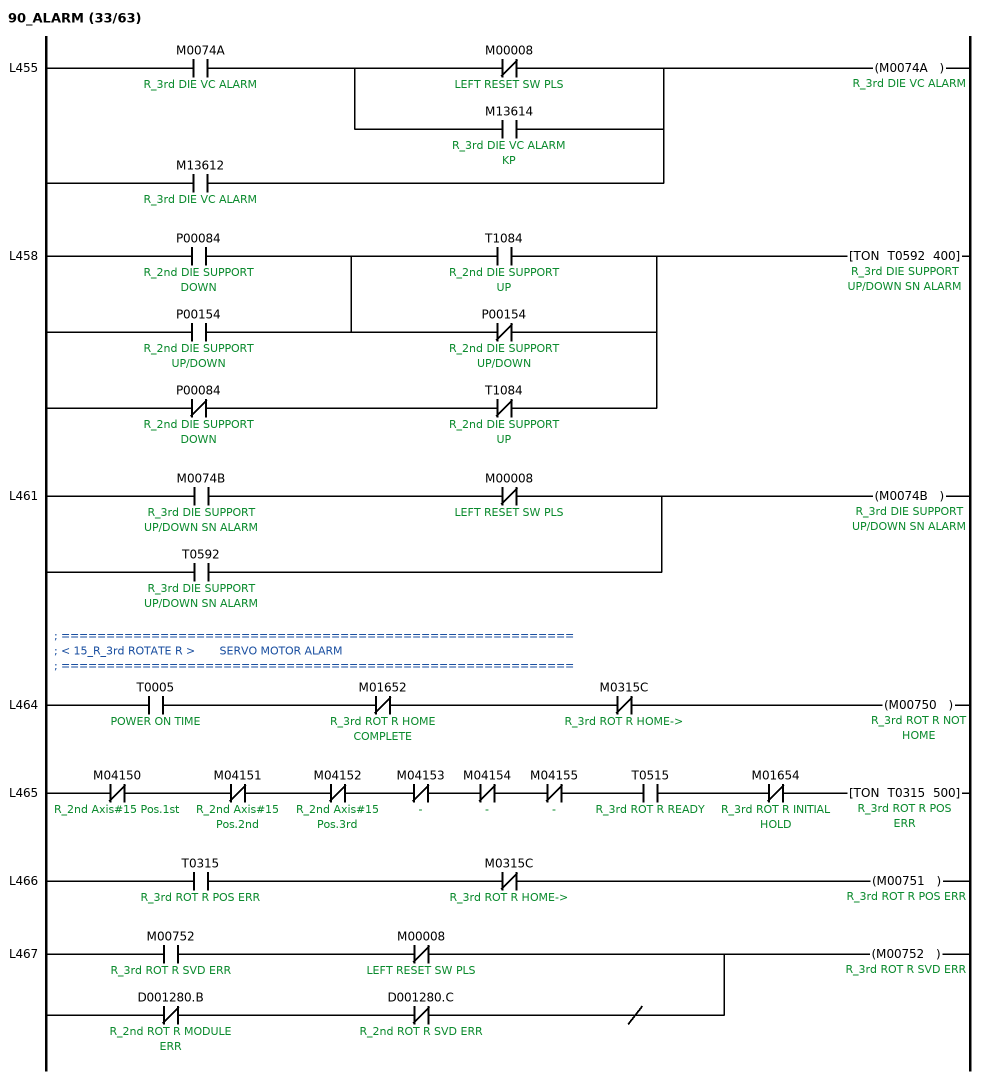
; L455
LOAD      M0074A	// R_3rd DIE VC ALARM
LOAD NOT  M00008	// LEFT RESET SW PLS
OR        M13614	// R_3rd DIE VC ALARM KP
AND LOAD
OR        M13612	// R_3rd DIE VC ALARM
OUT       M0074A	// R_3rd DIE VC ALARM
; L458
LOAD      P00084	// R_2nd DIE SUPPORT DOWN
OR        P00154	// R_2nd DIE SUPPORT UP/DOWN
LOAD      T1084	// R_2nd DIE SUPPORT UP
OR NOT    P00154	// R_2nd DIE SUPPORT UP/DOWN
AND LOAD
LOAD NOT  P00084	// R_2nd DIE SUPPORT DOWN
AND NOT   T1084	// R_2nd DIE SUPPORT UP
OR LOAD
TON       T0592 400	// R_3rd DIE SUPPORT UP/DOWN SN ALARM
; L461
LOAD      M0074B	// R_3rd DIE SUPPORT UP/DOWN SN ALARM
AND NOT   M00008	// LEFT RESET SW PLS
OR        T0592	// R_3rd DIE SUPPORT UP/DOWN SN ALARM
OUT       M0074B	// R_3rd DIE SUPPORT UP/DOWN SN ALARM
// =========================================================
// 
//        < 15_R_3rd ROTATE R >       SERVO MOTOR ALARM
// 
// =========================================================
; L464
LOAD      T0005	// POWER ON TIME
AND NOT   M01652	// R_3rd ROT R HOME COMPLETE
AND NOT   M0315C	// R_3rd ROT R HOME->
OUT       M00750	// R_3rd ROT R NOT HOME
; L465
LOAD NOT  M04150	// R_2nd Axis#15 Pos.1st
AND NOT   M04151	// R_2nd Axis#15 Pos.2nd
AND NOT   M04152	// R_2nd Axis#15 Pos.3rd
AND NOT   M04153	// -
AND NOT   M04154	// -
AND NOT   M04155	// -
AND       T0515	// R_3rd ROT R READY
AND NOT   M01654	// R_3rd ROT R INITIAL HOLD
TON       T0315 500	// R_3rd ROT R POS ERR
; L466
LOAD      T0315	// R_3rd ROT R POS ERR
AND NOT   M0315C	// R_3rd ROT R HOME->
OUT       M00751	// R_3rd ROT R POS ERR
; L467
LOAD      M00752	// R_3rd ROT R SVD ERR
AND NOT   M00008	// LEFT RESET SW PLS
LOAD NOT  D001280.B	// R_2nd ROT R MODULE ERR
AND NOT   D001280.C	// R_2nd ROT R SVD ERR
NOT
OR LOAD
OUT       M00752	// R_3rd ROT R SVD ERR

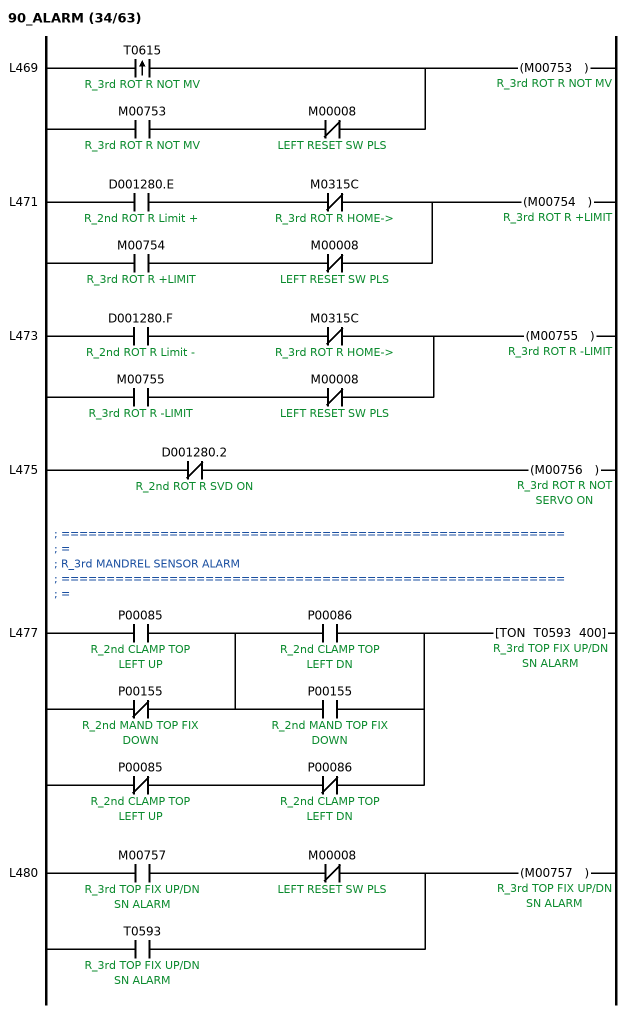
; L469
LOADP     T0615	// R_3rd ROT R NOT MV
LOAD      M00753	// R_3rd ROT R NOT MV
AND NOT   M00008	// LEFT RESET SW PLS
OR LOAD
OUT       M00753	// R_3rd ROT R NOT MV
; L471
LOAD      D001280.E	// R_2nd ROT R Limit +
AND NOT   M0315C	// R_3rd ROT R HOME->
LOAD      M00754	// R_3rd ROT R +LIMIT
AND NOT   M00008	// LEFT RESET SW PLS
OR LOAD
OUT       M00754	// R_3rd ROT R +LIMIT
; L473
LOAD      D001280.F	// R_2nd ROT R Limit -
AND NOT   M0315C	// R_3rd ROT R HOME->
LOAD      M00755	// R_3rd ROT R -LIMIT
AND NOT   M00008	// LEFT RESET SW PLS
OR LOAD
OUT       M00755	// R_3rd ROT R -LIMIT
; L475
LOAD NOT  D001280.2	// R_2nd ROT R SVD ON
OUT       M00756	// R_3rd ROT R NOT SERVO ON
// =========================================================
// 
//        R_3rd MANDREL SENSOR ALARM
// 
// =========================================================
; L477
LOAD      P00085	// R_2nd CLAMP TOP LEFT UP
OR NOT    P00155	// R_2nd MAND TOP FIX DOWN
LOAD      P00086	// R_2nd CLAMP TOP LEFT DN
OR        P00155	// R_2nd MAND TOP FIX DOWN
AND LOAD
LOAD NOT  P00085	// R_2nd CLAMP TOP LEFT UP
AND NOT   P00086	// R_2nd CLAMP TOP LEFT DN
OR LOAD
TON       T0593 400	// R_3rd TOP FIX UP/DN SN ALARM
; L480
LOAD      M00757	// R_3rd TOP FIX UP/DN SN ALARM
AND NOT   M00008	// LEFT RESET SW PLS
OR        T0593	// R_3rd TOP FIX UP/DN SN ALARM
OUT       M00757	// R_3rd TOP FIX UP/DN SN ALARM

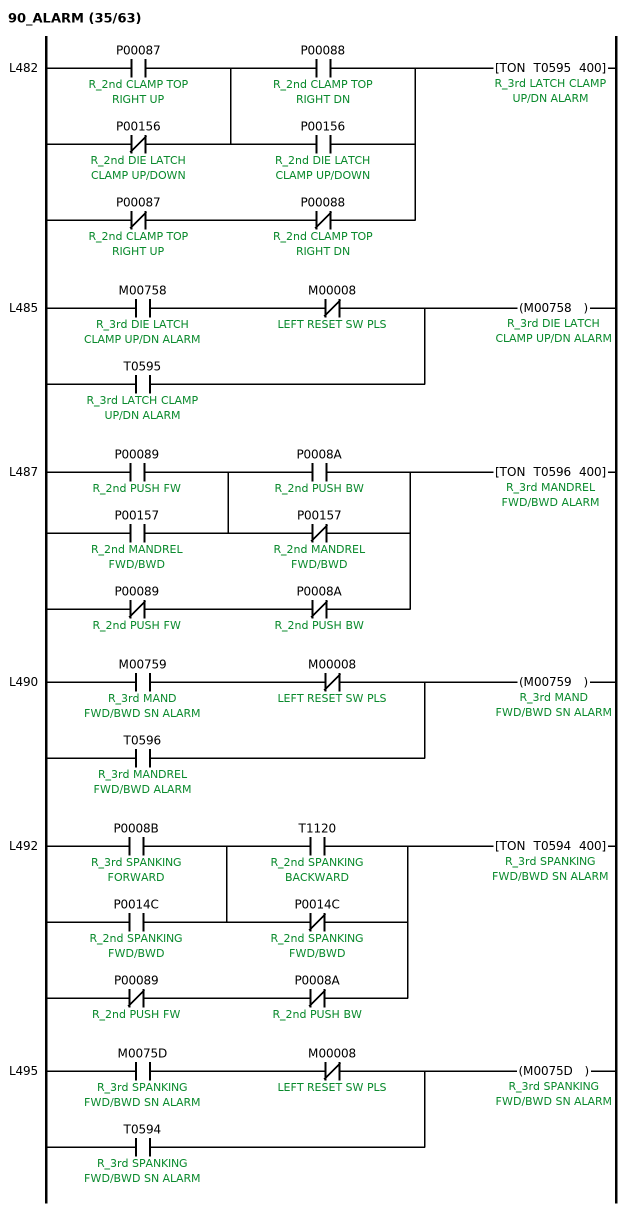
; L482
LOAD      P00087	// R_2nd CLAMP TOP RIGHT UP
OR NOT    P00156	// R_2nd DIE LATCH CLAMP UP/DOWN
LOAD      P00088	// R_2nd CLAMP TOP RIGHT DN
OR        P00156	// R_2nd DIE LATCH CLAMP UP/DOWN
AND LOAD
LOAD NOT  P00087	// R_2nd CLAMP TOP RIGHT UP
AND NOT   P00088	// R_2nd CLAMP TOP RIGHT DN
OR LOAD
TON       T0595 400	// R_3rd LATCH CLAMP UP/DN ALARM
; L485
LOAD      M00758	// R_3rd DIE LATCH CLAMP UP/DN ALARM
AND NOT   M00008	// LEFT RESET SW PLS
OR        T0595	// R_3rd LATCH CLAMP UP/DN ALARM
OUT       M00758	// R_3rd DIE LATCH CLAMP UP/DN ALARM
; L487
LOAD      P00089	// R_2nd PUSH FW
OR        P00157	// R_2nd MANDREL FWD/BWD
LOAD      P0008A	// R_2nd PUSH BW
OR NOT    P00157	// R_2nd MANDREL FWD/BWD
AND LOAD
LOAD NOT  P00089	// R_2nd PUSH FW
AND NOT   P0008A	// R_2nd PUSH BW
OR LOAD
TON       T0596 400	// R_3rd MANDREL FWD/BWD ALARM
; L490
LOAD      M00759	// R_3rd MAND FWD/BWD SN ALARM
AND NOT   M00008	// LEFT RESET SW PLS
OR        T0596	// R_3rd MANDREL FWD/BWD ALARM
OUT       M00759	// R_3rd MAND FWD/BWD SN ALARM
; L492
LOAD      P0008B	// R_3rd SPANKING FORWARD
OR        P0014C	// R_2nd SPANKING FWD/BWD
LOAD      T1120	// R_2nd SPANKING BACKWARD
OR NOT    P0014C	// R_2nd SPANKING FWD/BWD
AND LOAD
LOAD NOT  P00089	// R_2nd PUSH FW
AND NOT   P0008A	// R_2nd PUSH BW
OR LOAD
TON       T0594 400	// R_3rd SPANKING FWD/BWD SN ALARM
; L495
LOAD      M0075D	// R_3rd SPANKING FWD/BWD SN ALARM
AND NOT   M00008	// LEFT RESET SW PLS
OR        T0594	// R_3rd SPANKING FWD/BWD SN ALARM
OUT       M0075D	// R_3rd SPANKING FWD/BWD SN ALARM

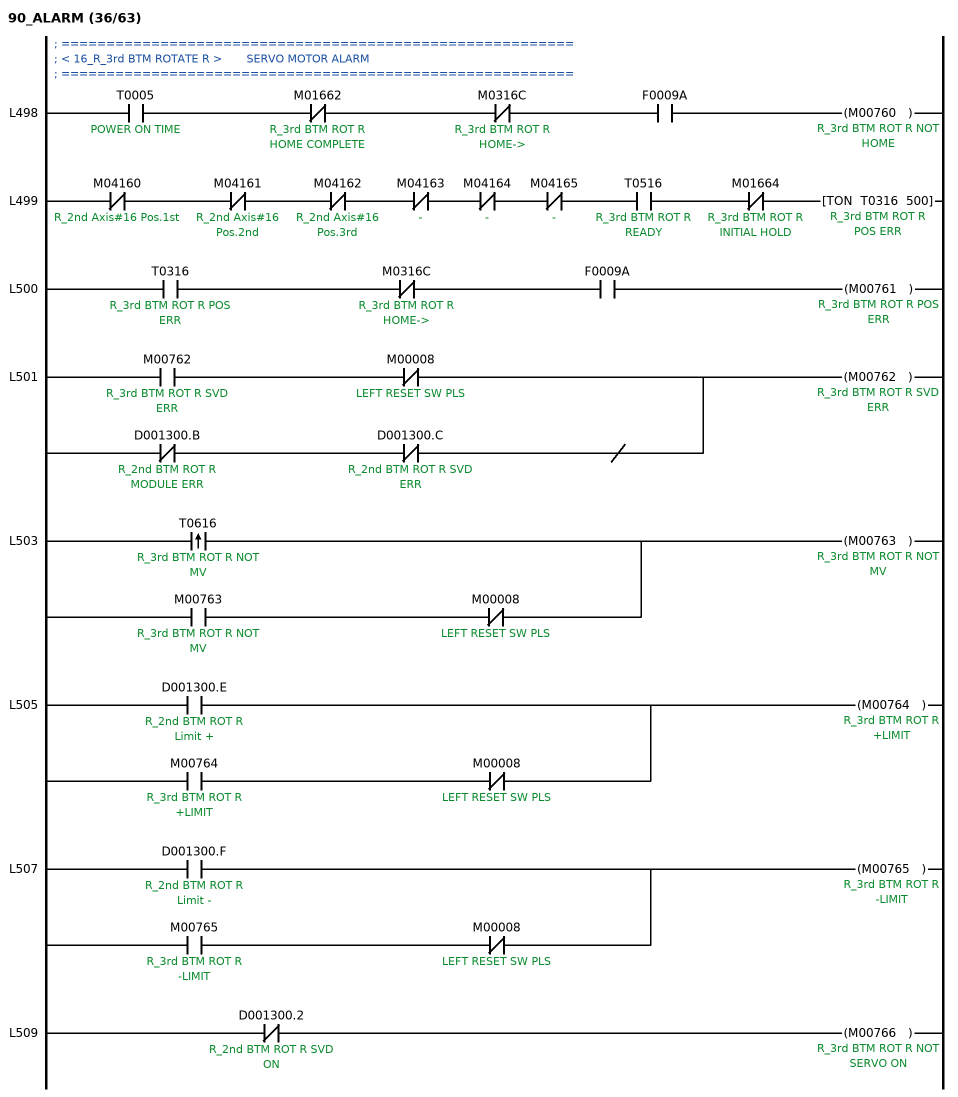
// =========================================================
// 
//        < 16_R_3rd BTM ROTATE R >       SERVO MOTOR ALARM
// 
// =========================================================
; L498
LOAD      T0005	// POWER ON TIME
AND NOT   M01662	// R_3rd BTM ROT R HOME COMPLETE
AND NOT   M0316C	// R_3rd BTM ROT R HOME->
AND       F0009A
OUT       M00760	// R_3rd BTM ROT R NOT HOME
; L499
LOAD NOT  M04160	// R_2nd Axis#16 Pos.1st
AND NOT   M04161	// R_2nd Axis#16 Pos.2nd
AND NOT   M04162	// R_2nd Axis#16 Pos.3rd
AND NOT   M04163	// -
AND NOT   M04164	// -
AND NOT   M04165	// -
AND       T0516	// R_3rd BTM ROT R READY
AND NOT   M01664	// R_3rd BTM ROT R INITIAL HOLD
TON       T0316 500	// R_3rd BTM ROT R POS ERR
; L500
LOAD      T0316	// R_3rd BTM ROT R POS ERR
AND NOT   M0316C	// R_3rd BTM ROT R HOME->
AND       F0009A
OUT       M00761	// R_3rd BTM ROT R POS ERR
; L501
LOAD      M00762	// R_3rd BTM ROT R SVD ERR
AND NOT   M00008	// LEFT RESET SW PLS
LOAD NOT  D001300.B	// R_2nd BTM ROT R MODULE ERR
AND NOT   D001300.C	// R_2nd BTM ROT R SVD ERR
NOT
OR LOAD
OUT       M00762	// R_3rd BTM ROT R SVD ERR
; L503
LOADP     T0616	// R_3rd BTM ROT R NOT MV
LOAD      M00763	// R_3rd BTM ROT R NOT MV
AND NOT   M00008	// LEFT RESET SW PLS
OR LOAD
OUT       M00763	// R_3rd BTM ROT R NOT MV
; L505
LOAD      D001300.E	// R_2nd BTM ROT R Limit +
LOAD      M00764	// R_3rd BTM ROT R +LIMIT
AND NOT   M00008	// LEFT RESET SW PLS
OR LOAD
OUT       M00764	// R_3rd BTM ROT R +LIMIT
; L507
LOAD      D001300.F	// R_2nd BTM ROT R Limit -
LOAD      M00765	// R_3rd BTM ROT R -LIMIT
AND NOT   M00008	// LEFT RESET SW PLS
OR LOAD
OUT       M00765	// R_3rd BTM ROT R -LIMIT
; L509
LOAD NOT  D001300.2	// R_2nd BTM ROT R SVD ON
OUT       M00766	// R_3rd BTM ROT R NOT SERVO ON

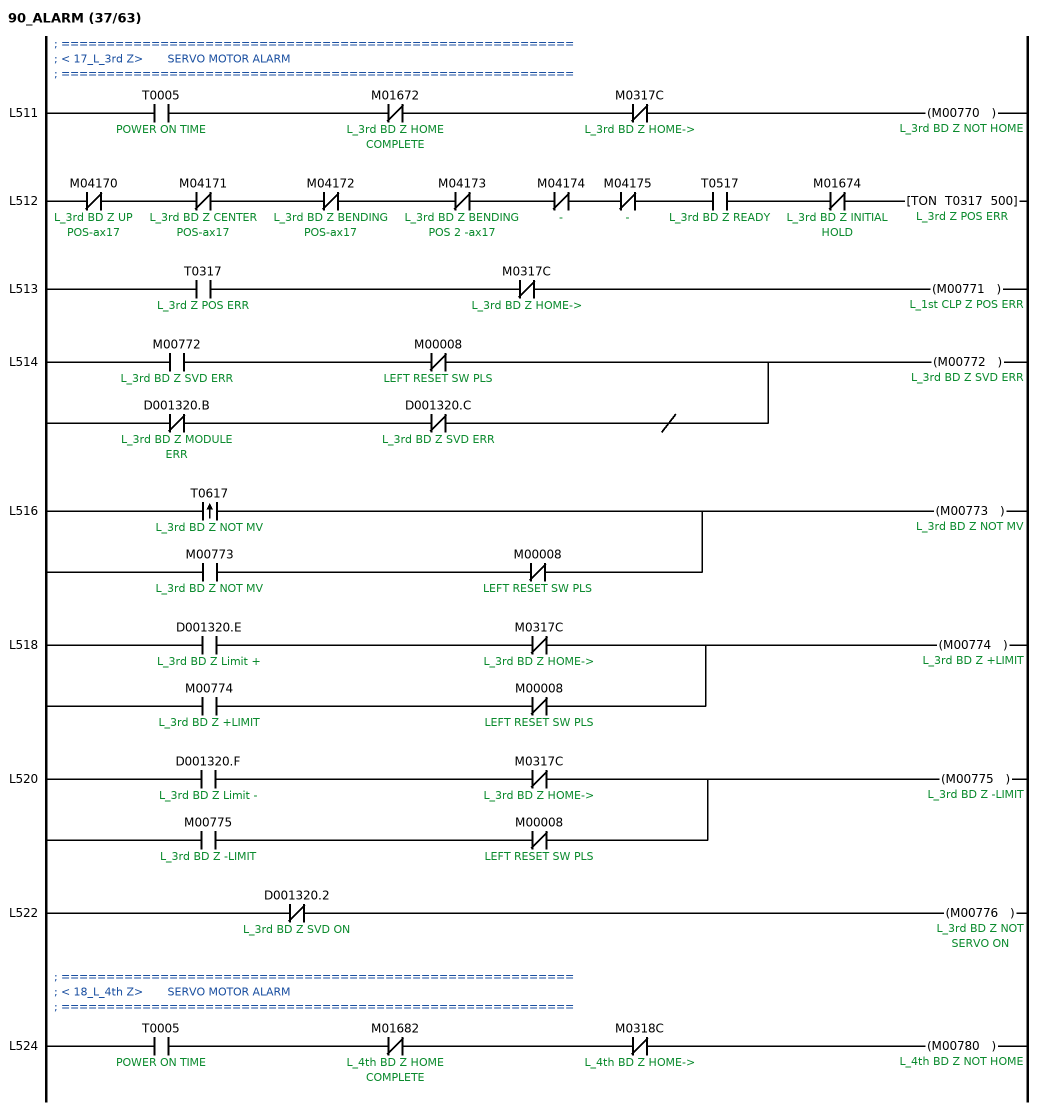
// =========================================================
// 
//        < 17_L_3rd Z>       SERVO MOTOR ALARM
// 
// =========================================================
; L511
LOAD      T0005	// POWER ON TIME
AND NOT   M01672	// L_3rd BD Z HOME COMPLETE
AND NOT   M0317C	// L_3rd BD Z HOME->
OUT       M00770	// L_3rd BD Z NOT HOME
; L512
LOAD NOT  M04170	// L_3rd BD Z UP POS-ax17
AND NOT   M04171	// L_3rd BD Z CENTER POS-ax17
AND NOT   M04172	// L_3rd BD Z BENDING POS-ax17
AND NOT   M04173	// L_3rd BD Z BENDING POS 2 -ax17
AND NOT   M04174	// -
AND NOT   M04175	// -
AND       T0517	// L_3rd BD Z READY
AND NOT   M01674	// L_3rd BD Z INITIAL HOLD
TON       T0317 500	// L_3rd Z POS ERR
; L513
LOAD      T0317	// L_3rd Z POS ERR
AND NOT   M0317C	// L_3rd BD Z HOME->
OUT       M00771	// L_1st CLP Z POS ERR
; L514
LOAD      M00772	// L_3rd BD Z SVD ERR
AND NOT   M00008	// LEFT RESET SW PLS
LOAD NOT  D001320.B	// L_3rd BD Z MODULE ERR
AND NOT   D001320.C	// L_3rd BD Z SVD ERR
NOT
OR LOAD
OUT       M00772	// L_3rd BD Z SVD ERR
; L516
LOADP     T0617	// L_3rd BD Z NOT MV
LOAD      M00773	// L_3rd BD Z NOT MV
AND NOT   M00008	// LEFT RESET SW PLS
OR LOAD
OUT       M00773	// L_3rd BD Z NOT MV
; L518
LOAD      D001320.E	// L_3rd BD Z Limit +
AND NOT   M0317C	// L_3rd BD Z HOME->
LOAD      M00774	// L_3rd BD Z +LIMIT
AND NOT   M00008	// LEFT RESET SW PLS
OR LOAD
OUT       M00774	// L_3rd BD Z +LIMIT
; L520
LOAD      D001320.F	// L_3rd BD Z Limit -
AND NOT   M0317C	// L_3rd BD Z HOME->
LOAD      M00775	// L_3rd BD Z -LIMIT
AND NOT   M00008	// LEFT RESET SW PLS
OR LOAD
OUT       M00775	// L_3rd BD Z -LIMIT
; L522
LOAD NOT  D001320.2	// L_3rd BD Z SVD ON
OUT       M00776	// L_3rd BD Z NOT SERVO ON
// =========================================================
// 
//        < 18_L_4th Z>       SERVO MOTOR ALARM
// 
// =========================================================
; L524
LOAD      T0005	// POWER ON TIME
AND NOT   M01682	// L_4th BD Z HOME COMPLETE
AND NOT   M0318C	// L_4th BD Z HOME->
OUT       M00780	// L_4th BD Z NOT HOME

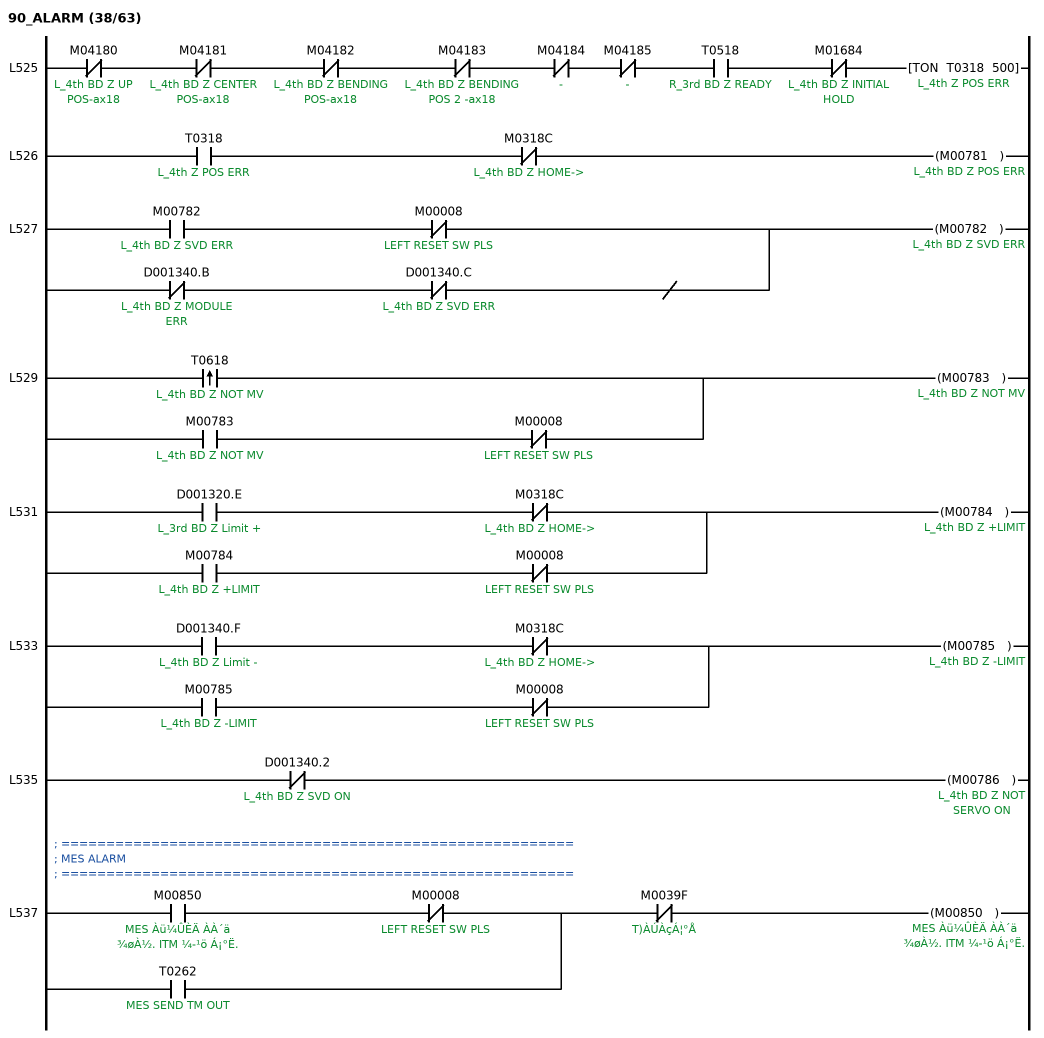
; L525
LOAD NOT  M04180	// L_4th BD Z UP POS-ax18
AND NOT   M04181	// L_4th BD Z CENTER POS-ax18
AND NOT   M04182	// L_4th BD Z BENDING POS-ax18
AND NOT   M04183	// L_4th BD Z BENDING POS 2 -ax18
AND NOT   M04184	// -
AND NOT   M04185	// -
AND       T0518	// R_3rd BD Z READY
AND NOT   M01684	// L_4th BD Z INITIAL HOLD
TON       T0318 500	// L_4th Z POS ERR
; L526
LOAD      T0318	// L_4th Z POS ERR
AND NOT   M0318C	// L_4th BD Z HOME->
OUT       M00781	// L_4th BD Z POS ERR
; L527
LOAD      M00782	// L_4th BD Z SVD ERR
AND NOT   M00008	// LEFT RESET SW PLS
LOAD NOT  D001340.B	// L_4th BD Z MODULE ERR
AND NOT   D001340.C	// L_4th BD Z SVD ERR
NOT
OR LOAD
OUT       M00782	// L_4th BD Z SVD ERR
; L529
LOADP     T0618	// L_4th BD Z NOT MV
LOAD      M00783	// L_4th BD Z NOT MV
AND NOT   M00008	// LEFT RESET SW PLS
OR LOAD
OUT       M00783	// L_4th BD Z NOT MV
; L531
LOAD      D001320.E	// L_3rd BD Z Limit +
AND NOT   M0318C	// L_4th BD Z HOME->
LOAD      M00784	// L_4th BD Z +LIMIT
AND NOT   M00008	// LEFT RESET SW PLS
OR LOAD
OUT       M00784	// L_4th BD Z +LIMIT
; L533
LOAD      D001340.F	// L_4th BD Z Limit -
AND NOT   M0318C	// L_4th BD Z HOME->
LOAD      M00785	// L_4th BD Z -LIMIT
AND NOT   M00008	// LEFT RESET SW PLS
OR LOAD
OUT       M00785	// L_4th BD Z -LIMIT
; L535
LOAD NOT  D001340.2	// L_4th BD Z SVD ON
OUT       M00786	// L_4th BD Z NOT SERVO ON
// =========================================================
// 
//        MES ALARM
// 
// =========================================================
; L537
LOAD      M00850	// MES Àü¼ÛÈÄ ÀÀ´ä ¾øÀ½. ITM ¼­¹ö Á¡°Ë.
AND NOT   M00008	// LEFT RESET SW PLS
OR        T0262	// MES SEND TM OUT
AND NOT   M0039F	// T)ÀÚÀçÁ¦°Å
OUT       M00850	// MES Àü¼ÛÈÄ ÀÀ´ä ¾øÀ½. ITM ¼­¹ö Á¡°Ë.

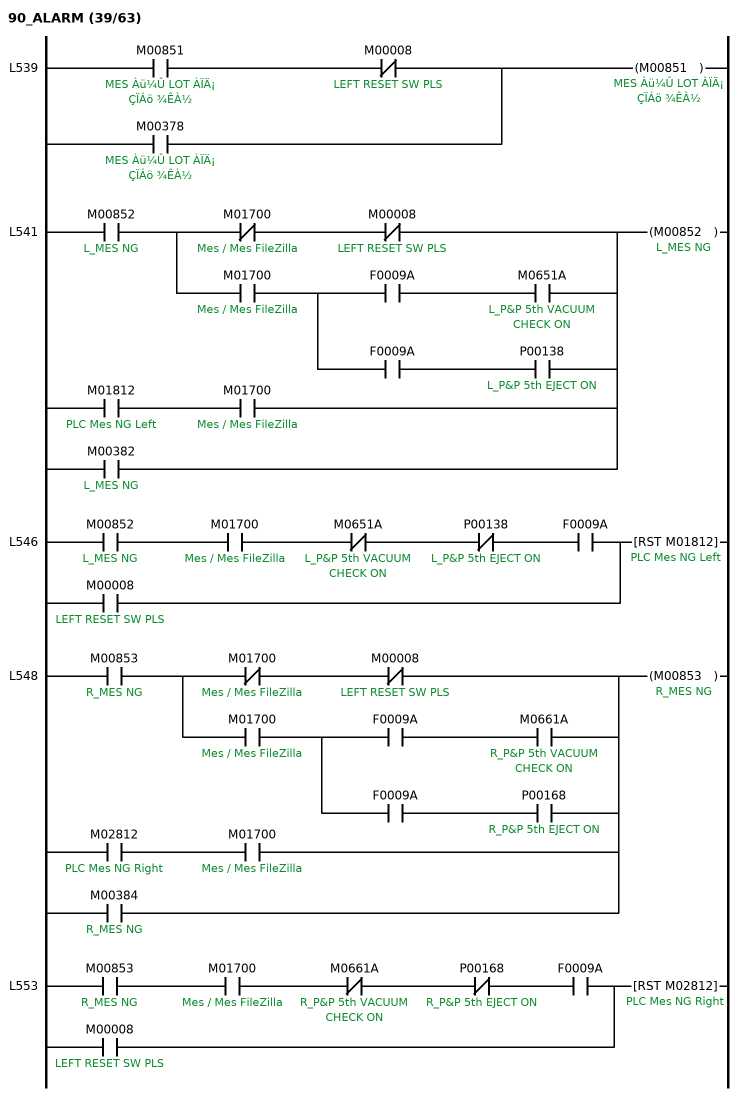
; L539
LOAD      M00851	// MES Àü¼Û LOT ÀÏÄ¡ ÇÏÁö ¾ÊÀ½
AND NOT   M00008	// LEFT RESET SW PLS
OR        M00378	// MES Àü¼Û LOT ÀÏÄ¡ ÇÏÁö ¾ÊÀ½
OUT       M00851	// MES Àü¼Û LOT ÀÏÄ¡ ÇÏÁö ¾ÊÀ½
; L541
LOAD      M00852	// L_MES NG
LOAD NOT  M01700	// Mes / Mes FileZilla
AND NOT   M00008	// LEFT RESET SW PLS
LOAD      M01700	// Mes / Mes FileZilla
LOAD      F0009A
AND       M0651A	// L_P&P 5th VACUUM CHECK ON
LOAD      F0009A
AND       P00138	// L_P&P 5th EJECT ON
OR LOAD
AND LOAD
OR LOAD
AND LOAD
LOAD      M01812	// PLC Mes NG Left
AND       M01700	// Mes / Mes FileZilla
OR LOAD
OR        M00382	// L_MES NG
OUT       M00852	// L_MES NG
; L546
LOAD      M00852	// L_MES NG
AND       M01700	// Mes / Mes FileZilla
AND NOT   M0651A	// L_P&P 5th VACUUM CHECK ON
AND NOT   P00138	// L_P&P 5th EJECT ON
AND       F0009A
OR        M00008	// LEFT RESET SW PLS
RST       M01812	// PLC Mes NG Left
; L548
LOAD      M00853	// R_MES NG
LOAD NOT  M01700	// Mes / Mes FileZilla
AND NOT   M00008	// LEFT RESET SW PLS
LOAD      M01700	// Mes / Mes FileZilla
LOAD      F0009A
AND       M0661A	// R_P&P 5th VACUUM CHECK ON
LOAD      F0009A
AND       P00168	// R_P&P 5th EJECT ON
OR LOAD
AND LOAD
OR LOAD
AND LOAD
LOAD      M02812	// PLC Mes NG Right
AND       M01700	// Mes / Mes FileZilla
OR LOAD
OR        M00384	// R_MES NG
OUT       M00853	// R_MES NG
; L553
LOAD      M00853	// R_MES NG
AND       M01700	// Mes / Mes FileZilla
AND NOT   M0661A	// R_P&P 5th VACUUM CHECK ON
AND NOT   P00168	// R_P&P 5th EJECT ON
AND       F0009A
OR        M00008	// LEFT RESET SW PLS
RST       M02812	// PLC Mes NG Right

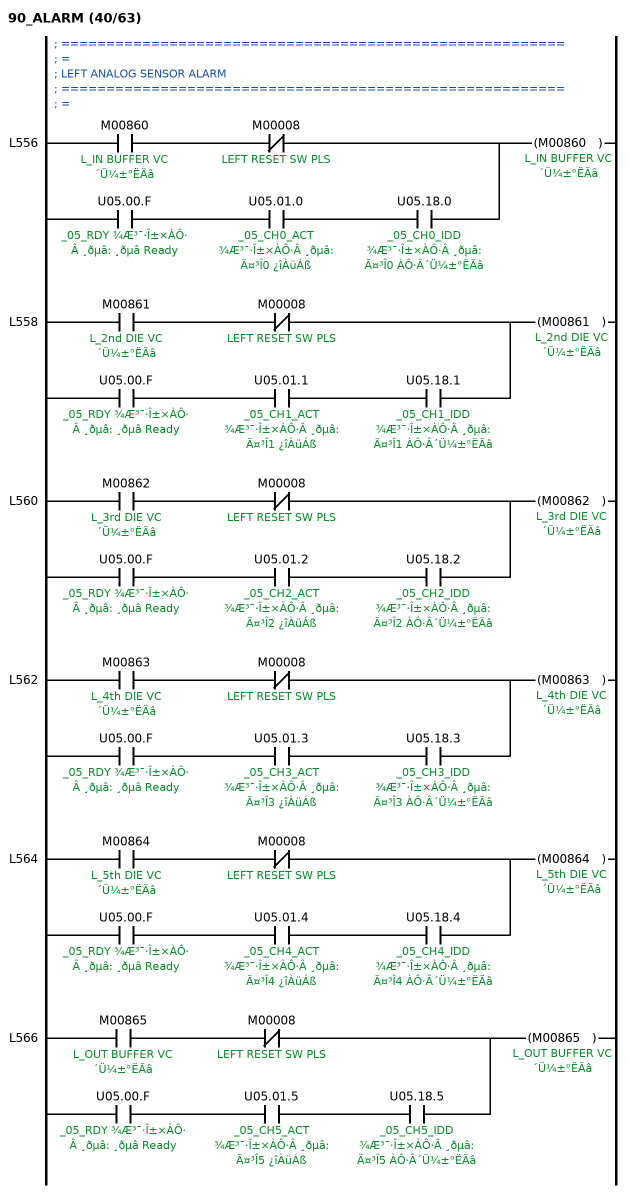
// =========================================================
// 
//        LEFT ANALOG SENSOR ALARM
// 
// =========================================================
; L556
LOAD      M00860	// L_IN BUFFER VC ´Ü¼±°ËÃâ
AND NOT   M00008	// LEFT RESET SW PLS
LOAD      U05.00.F	// _05_RDY ¾Æ³¯·Î±×ÀÔ·Â ¸ðµâ: ¸ðµâ Ready
AND       U05.01.0	// _05_CH0_ACT ¾Æ³¯·Î±×ÀÔ·Â ¸ðµâ: Ã¤³Î0 ¿îÀüÁß
AND       U05.18.0	// _05_CH0_IDD ¾Æ³¯·Î±×ÀÔ·Â ¸ðµâ: Ã¤³Î0 ÀÔ·Â´Ü¼±°ËÃâ
OR LOAD
OUT       M00860	// L_IN BUFFER VC ´Ü¼±°ËÃâ
; L558
LOAD      M00861	// L_2nd DIE VC ´Ü¼±°ËÃâ
AND NOT   M00008	// LEFT RESET SW PLS
LOAD      U05.00.F	// _05_RDY ¾Æ³¯·Î±×ÀÔ·Â ¸ðµâ: ¸ðµâ Ready
AND       U05.01.1	// _05_CH1_ACT ¾Æ³¯·Î±×ÀÔ·Â ¸ðµâ: Ã¤³Î1 ¿îÀüÁß
AND       U05.18.1	// _05_CH1_IDD ¾Æ³¯·Î±×ÀÔ·Â ¸ðµâ: Ã¤³Î1 ÀÔ·Â´Ü¼±°ËÃâ
OR LOAD
OUT       M00861	// L_2nd DIE VC ´Ü¼±°ËÃâ
; L560
LOAD      M00862	// L_3rd DIE VC ´Ü¼±°ËÃâ
AND NOT   M00008	// LEFT RESET SW PLS
LOAD      U05.00.F	// _05_RDY ¾Æ³¯·Î±×ÀÔ·Â ¸ðµâ: ¸ðµâ Ready
AND       U05.01.2	// _05_CH2_ACT ¾Æ³¯·Î±×ÀÔ·Â ¸ðµâ: Ã¤³Î2 ¿îÀüÁß
AND       U05.18.2	// _05_CH2_IDD ¾Æ³¯·Î±×ÀÔ·Â ¸ðµâ: Ã¤³Î2 ÀÔ·Â´Ü¼±°ËÃâ
OR LOAD
OUT       M00862	// L_3rd DIE VC ´Ü¼±°ËÃâ
; L562
LOAD      M00863	// L_4th DIE VC ´Ü¼±°ËÃâ
AND NOT   M00008	// LEFT RESET SW PLS
LOAD      U05.00.F	// _05_RDY ¾Æ³¯·Î±×ÀÔ·Â ¸ðµâ: ¸ðµâ Ready
AND       U05.01.3	// _05_CH3_ACT ¾Æ³¯·Î±×ÀÔ·Â ¸ðµâ: Ã¤³Î3 ¿îÀüÁß
AND       U05.18.3	// _05_CH3_IDD ¾Æ³¯·Î±×ÀÔ·Â ¸ðµâ: Ã¤³Î3 ÀÔ·Â´Ü¼±°ËÃâ
OR LOAD
OUT       M00863	// L_4th DIE VC ´Ü¼±°ËÃâ
; L564
LOAD      M00864	// L_5th DIE VC ´Ü¼±°ËÃâ
AND NOT   M00008	// LEFT RESET SW PLS
LOAD      U05.00.F	// _05_RDY ¾Æ³¯·Î±×ÀÔ·Â ¸ðµâ: ¸ðµâ Ready
AND       U05.01.4	// _05_CH4_ACT ¾Æ³¯·Î±×ÀÔ·Â ¸ðµâ: Ã¤³Î4 ¿îÀüÁß
AND       U05.18.4	// _05_CH4_IDD ¾Æ³¯·Î±×ÀÔ·Â ¸ðµâ: Ã¤³Î4 ÀÔ·Â´Ü¼±°ËÃâ
OR LOAD
OUT       M00864	// L_5th DIE VC ´Ü¼±°ËÃâ
; L566
LOAD      M00865	// L_OUT BUFFER VC ´Ü¼±°ËÃâ
AND NOT   M00008	// LEFT RESET SW PLS
LOAD      U05.00.F	// _05_RDY ¾Æ³¯·Î±×ÀÔ·Â ¸ðµâ: ¸ðµâ Ready
AND       U05.01.5	// _05_CH5_ACT ¾Æ³¯·Î±×ÀÔ·Â ¸ðµâ: Ã¤³Î5 ¿îÀüÁß
AND       U05.18.5	// _05_CH5_IDD ¾Æ³¯·Î±×ÀÔ·Â ¸ðµâ: Ã¤³Î5 ÀÔ·Â´Ü¼±°ËÃâ
OR LOAD
OUT       M00865	// L_OUT BUFFER VC ´Ü¼±°ËÃâ

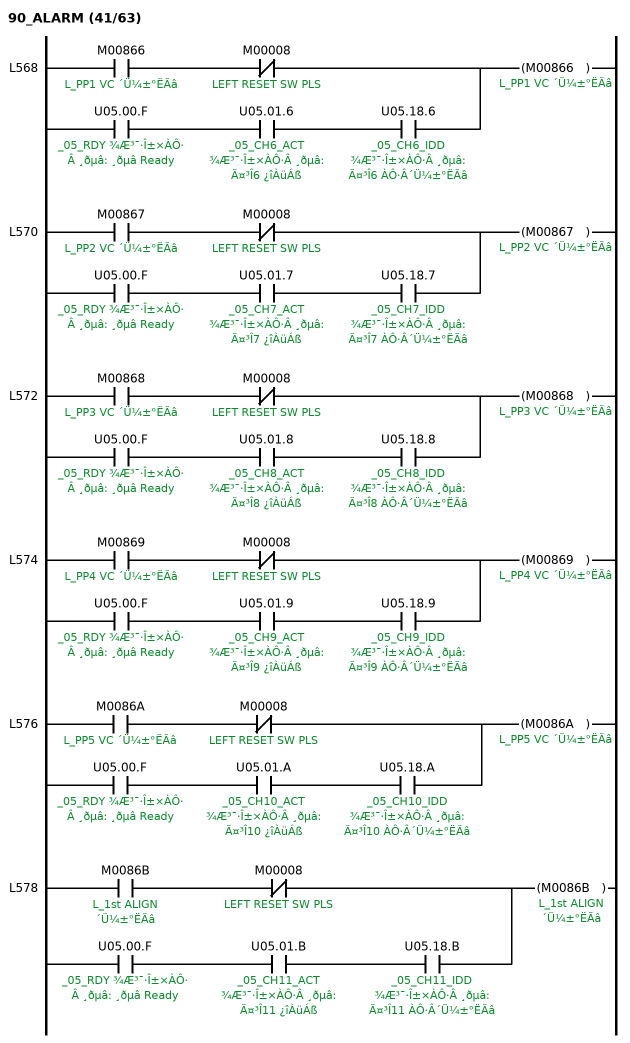
; L568
LOAD      M00866	// L_PP1 VC ´Ü¼±°ËÃâ
AND NOT   M00008	// LEFT RESET SW PLS
LOAD      U05.00.F	// _05_RDY ¾Æ³¯·Î±×ÀÔ·Â ¸ðµâ: ¸ðµâ Ready
AND       U05.01.6	// _05_CH6_ACT ¾Æ³¯·Î±×ÀÔ·Â ¸ðµâ: Ã¤³Î6 ¿îÀüÁß
AND       U05.18.6	// _05_CH6_IDD ¾Æ³¯·Î±×ÀÔ·Â ¸ðµâ: Ã¤³Î6 ÀÔ·Â´Ü¼±°ËÃâ
OR LOAD
OUT       M00866	// L_PP1 VC ´Ü¼±°ËÃâ
; L570
LOAD      M00867	// L_PP2 VC ´Ü¼±°ËÃâ
AND NOT   M00008	// LEFT RESET SW PLS
LOAD      U05.00.F	// _05_RDY ¾Æ³¯·Î±×ÀÔ·Â ¸ðµâ: ¸ðµâ Ready
AND       U05.01.7	// _05_CH7_ACT ¾Æ³¯·Î±×ÀÔ·Â ¸ðµâ: Ã¤³Î7 ¿îÀüÁß
AND       U05.18.7	// _05_CH7_IDD ¾Æ³¯·Î±×ÀÔ·Â ¸ðµâ: Ã¤³Î7 ÀÔ·Â´Ü¼±°ËÃâ
OR LOAD
OUT       M00867	// L_PP2 VC ´Ü¼±°ËÃâ
; L572
LOAD      M00868	// L_PP3 VC ´Ü¼±°ËÃâ
AND NOT   M00008	// LEFT RESET SW PLS
LOAD      U05.00.F	// _05_RDY ¾Æ³¯·Î±×ÀÔ·Â ¸ðµâ: ¸ðµâ Ready
AND       U05.01.8	// _05_CH8_ACT ¾Æ³¯·Î±×ÀÔ·Â ¸ðµâ: Ã¤³Î8 ¿îÀüÁß
AND       U05.18.8	// _05_CH8_IDD ¾Æ³¯·Î±×ÀÔ·Â ¸ðµâ: Ã¤³Î8 ÀÔ·Â´Ü¼±°ËÃâ
OR LOAD
OUT       M00868	// L_PP3 VC ´Ü¼±°ËÃâ
; L574
LOAD      M00869	// L_PP4 VC ´Ü¼±°ËÃâ
AND NOT   M00008	// LEFT RESET SW PLS
LOAD      U05.00.F	// _05_RDY ¾Æ³¯·Î±×ÀÔ·Â ¸ðµâ: ¸ðµâ Ready
AND       U05.01.9	// _05_CH9_ACT ¾Æ³¯·Î±×ÀÔ·Â ¸ðµâ: Ã¤³Î9 ¿îÀüÁß
AND       U05.18.9	// _05_CH9_IDD ¾Æ³¯·Î±×ÀÔ·Â ¸ðµâ: Ã¤³Î9 ÀÔ·Â´Ü¼±°ËÃâ
OR LOAD
OUT       M00869	// L_PP4 VC ´Ü¼±°ËÃâ
; L576
LOAD      M0086A	// L_PP5 VC ´Ü¼±°ËÃâ
AND NOT   M00008	// LEFT RESET SW PLS
LOAD      U05.00.F	// _05_RDY ¾Æ³¯·Î±×ÀÔ·Â ¸ðµâ: ¸ðµâ Ready
AND       U05.01.A	// _05_CH10_ACT ¾Æ³¯·Î±×ÀÔ·Â ¸ðµâ: Ã¤³Î10 ¿îÀüÁß
AND       U05.18.A	// _05_CH10_IDD ¾Æ³¯·Î±×ÀÔ·Â ¸ðµâ: Ã¤³Î10 ÀÔ·Â´Ü¼±°ËÃâ
OR LOAD
OUT       M0086A	// L_PP5 VC ´Ü¼±°ËÃâ
; L578
LOAD      M0086B	// L_1st ALIGN ´Ü¼±°ËÃâ
AND NOT   M00008	// LEFT RESET SW PLS
LOAD      U05.00.F	// _05_RDY ¾Æ³¯·Î±×ÀÔ·Â ¸ðµâ: ¸ðµâ Ready
AND       U05.01.B	// _05_CH11_ACT ¾Æ³¯·Î±×ÀÔ·Â ¸ðµâ: Ã¤³Î11 ¿îÀüÁß
AND       U05.18.B	// _05_CH11_IDD ¾Æ³¯·Î±×ÀÔ·Â ¸ðµâ: Ã¤³Î11 ÀÔ·Â´Ü¼±°ËÃâ
OR LOAD
OUT       M0086B	// L_1st ALIGN ´Ü¼±°ËÃâ

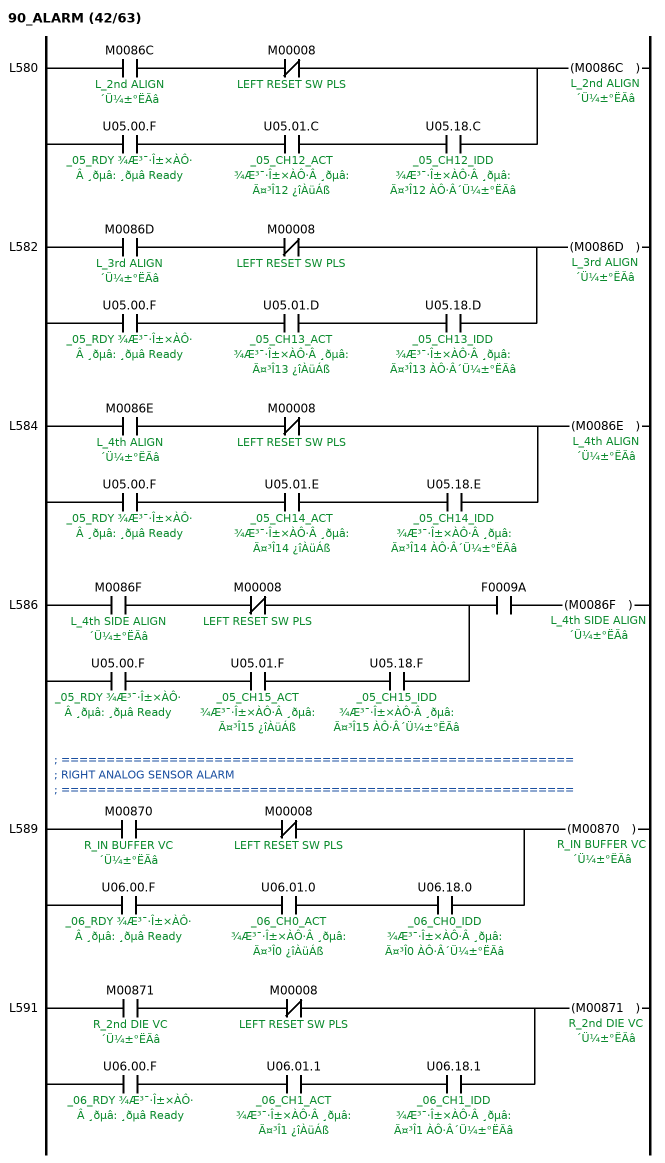
; L580
LOAD      M0086C	// L_2nd ALIGN ´Ü¼±°ËÃâ
AND NOT   M00008	// LEFT RESET SW PLS
LOAD      U05.00.F	// _05_RDY ¾Æ³¯·Î±×ÀÔ·Â ¸ðµâ: ¸ðµâ Ready
AND       U05.01.C	// _05_CH12_ACT ¾Æ³¯·Î±×ÀÔ·Â ¸ðµâ: Ã¤³Î12 ¿îÀüÁß
AND       U05.18.C	// _05_CH12_IDD ¾Æ³¯·Î±×ÀÔ·Â ¸ðµâ: Ã¤³Î12 ÀÔ·Â´Ü¼±°ËÃâ
OR LOAD
OUT       M0086C	// L_2nd ALIGN ´Ü¼±°ËÃâ
; L582
LOAD      M0086D	// L_3rd ALIGN ´Ü¼±°ËÃâ
AND NOT   M00008	// LEFT RESET SW PLS
LOAD      U05.00.F	// _05_RDY ¾Æ³¯·Î±×ÀÔ·Â ¸ðµâ: ¸ðµâ Ready
AND       U05.01.D	// _05_CH13_ACT ¾Æ³¯·Î±×ÀÔ·Â ¸ðµâ: Ã¤³Î13 ¿îÀüÁß
AND       U05.18.D	// _05_CH13_IDD ¾Æ³¯·Î±×ÀÔ·Â ¸ðµâ: Ã¤³Î13 ÀÔ·Â´Ü¼±°ËÃâ
OR LOAD
OUT       M0086D	// L_3rd ALIGN ´Ü¼±°ËÃâ
; L584
LOAD      M0086E	// L_4th ALIGN ´Ü¼±°ËÃâ
AND NOT   M00008	// LEFT RESET SW PLS
LOAD      U05.00.F	// _05_RDY ¾Æ³¯·Î±×ÀÔ·Â ¸ðµâ: ¸ðµâ Ready
AND       U05.01.E	// _05_CH14_ACT ¾Æ³¯·Î±×ÀÔ·Â ¸ðµâ: Ã¤³Î14 ¿îÀüÁß
AND       U05.18.E	// _05_CH14_IDD ¾Æ³¯·Î±×ÀÔ·Â ¸ðµâ: Ã¤³Î14 ÀÔ·Â´Ü¼±°ËÃâ
OR LOAD
OUT       M0086E	// L_4th ALIGN ´Ü¼±°ËÃâ
; L586
LOAD      M0086F	// L_4th SIDE ALIGN ´Ü¼±°ËÃâ
AND NOT   M00008	// LEFT RESET SW PLS
LOAD      U05.00.F	// _05_RDY ¾Æ³¯·Î±×ÀÔ·Â ¸ðµâ: ¸ðµâ Ready
AND       U05.01.F	// _05_CH15_ACT ¾Æ³¯·Î±×ÀÔ·Â ¸ðµâ: Ã¤³Î15 ¿îÀüÁß
AND       U05.18.F	// _05_CH15_IDD ¾Æ³¯·Î±×ÀÔ·Â ¸ðµâ: Ã¤³Î15 ÀÔ·Â´Ü¼±°ËÃâ
OR LOAD
AND       F0009A
OUT       M0086F	// L_4th SIDE ALIGN ´Ü¼±°ËÃâ
// =========================================================
// 
//        RIGHT ANALOG SENSOR ALARM
// 
// =========================================================
; L589
LOAD      M00870	// R_IN BUFFER VC ´Ü¼±°ËÃâ
AND NOT   M00008	// LEFT RESET SW PLS
LOAD      U06.00.F	// _06_RDY ¾Æ³¯·Î±×ÀÔ·Â ¸ðµâ: ¸ðµâ Ready
AND       U06.01.0	// _06_CH0_ACT ¾Æ³¯·Î±×ÀÔ·Â ¸ðµâ: Ã¤³Î0 ¿îÀüÁß
AND       U06.18.0	// _06_CH0_IDD ¾Æ³¯·Î±×ÀÔ·Â ¸ðµâ: Ã¤³Î0 ÀÔ·Â´Ü¼±°ËÃâ
OR LOAD
OUT       M00870	// R_IN BUFFER VC ´Ü¼±°ËÃâ
; L591
LOAD      M00871	// R_2nd DIE VC ´Ü¼±°ËÃâ
AND NOT   M00008	// LEFT RESET SW PLS
LOAD      U06.00.F	// _06_RDY ¾Æ³¯·Î±×ÀÔ·Â ¸ðµâ: ¸ðµâ Ready
AND       U06.01.1	// _06_CH1_ACT ¾Æ³¯·Î±×ÀÔ·Â ¸ðµâ: Ã¤³Î1 ¿îÀüÁß
AND       U06.18.1	// _06_CH1_IDD ¾Æ³¯·Î±×ÀÔ·Â ¸ðµâ: Ã¤³Î1 ÀÔ·Â´Ü¼±°ËÃâ
OR LOAD
OUT       M00871	// R_2nd DIE VC ´Ü¼±°ËÃâ

